FUNCTION_BLOCK "A0301_Spintore_Lat_FB"   // FB59, LAD
TITLE = == GESTIONE DELLA STAZIONE P5 ==
// stored: MemoryReserve 100, SetENOAutomatically false
   VAR_INPUT
      AreaInterface { ExternalAccessible := 'False'; ExternalVisible := 'False'; ExternalWritable := 'False'} : "AreaInterface";
      ZSI { ExternalAccessible := 'False'; ExternalVisible := 'False'; ExternalWritable := 'False'} : "udt_ZoneSafetyInterface";
      DSI { ExternalAccessible := 'False'; ExternalVisible := 'False'; ExternalWritable := 'False'} : "udt_DeviceSafetyInterface";
      DataIn : Struct
         OP_Rest_PB : Bool;
         OP_Work_PB : Bool;
         Orz_1_AnalSens : Int;
         Orz_2_AnalSens : Int;
      END_STRUCT;
      CIn { ExternalAccessible := 'False'; ExternalVisible := 'False'; ExternalWritable := 'False'} : Struct
         Manager_SpinLat_1 : "ValveMachine_Manager";
         Manager_SpinLat_2 : "ValveMachine_Manager";
         Manager_Sollevatori : "ValveMachine_Manager";
         SemiAut_Pb : Bool;
         P4 : Struct
            Fermi : "ValveMachine_COut";
         END_STRUCT;
         P5 : Struct
            SpintoreLong : Struct   // Spintore Longitudinale
               Ax_Sts : Struct
                  PosAttesa_Reached : Bool;
                  PosFineSpinta_Reached : Bool;
               END_STRUCT;
               Spintore : "ValveMachine_COut";
               Ax : "Positioning_EPOS_Machine_COut";
               Vrt : "ValveMachine_COut";
               Orz : "ValveMachine_COut";
            END_STRUCT;
         END_STRUCT;
         Trasporto : "SpeedMachine_COut";
      END_STRUCT;
      Config : Struct
         Vrt_1 : "ValveMachine_Config";
         Orz_1 : "ValveMachine_Config";
         Vrt_2 : "ValveMachine_Config";
         Orz_2 : "ValveMachine_Config";
         Sollevatori : Array[1..7] of "ValveMachine_Config";
         QuotaIngombro_SpinLat2 : Real := 2700.0;
         QuotaIngombro_SpinLat1 { ExternalWritable := 'False'} : Real := 770.0;
         DelayMissingCondition : Time;
      END_STRUCT;
   END_VAR
   VAR_OUTPUT
      MachineInterface : "MachineInterface";
      COut : Struct
         Spin_Lat1 : Struct
            Standstill : Bool;
            Rest_CheckNext : Bool;
            Work_CheckNext : Bool;
            Rest : Bool;
            Work : Bool;
         END_STRUCT;
         Spin_Lat2 : Struct
            Standstill : Bool;
            Rest_CheckNext : Bool;
            Work_CheckNext : Bool;
            Rest : Bool;
            Work : Bool;
         END_STRUCT;
         Vrt_1 : "ValveMachine_COut";
         Orz_1 : "ValveMachine_COut";
         Vrt_2 : "ValveMachine_COut";
         Orz_2 : "ValveMachine_COut";
         Sollevatori : "ValveMachine_COut";
      END_STRUCT;
   END_VAR
   VAR_IN_OUT
      Spin_Lat_1 : Struct
         Par : "Analogic_SensorManagement_Par";
         Data : Struct
            Sens : "Analogic_SensorManagement_Data";
            HMI : "HMI_Preset";
         END_STRUCT;
         Par_Mach : "A0301_Mach_Sens_Par";
      END_STRUCT;
      Spin_Lat_2 : Struct
         Par : "Analogic_SensorManagement_Par";
         Data : Struct
            Sens : "Analogic_SensorManagement_Data";
            HMI : "HMI_Preset";
         END_STRUCT;
         Par_Mach : "A0301_Mach_Sens_Par";
      END_STRUCT;
   END_VAR
   VAR
      Alarm : Struct
         Vrt_1 : "ValveAlr";
         Orz_1 { S7_SetPoint := 'True'} : "ValveAlr";
         Orz_1_AnalSens_Issue : Bool;
         Vrt_2 : "ValveAlr";
         Orz_2 { S7_SetPoint := 'True'} : "ValveAlr";
         Orz_2_AnalSens_Issue : Bool;
         Sollevatori : Array[1..7] of "ValveAlr";
         Finestre : Struct
            SpinLat2_SpinLong_Stop : Bool;   // Allarme Spintore longitudinale a ridosso dello Spintore laterale 2 che non si è abbassato
            SpinLat1_SpinLong_Stop : Bool;   // Allarme Spintore longitudinale a ridosso dello Spintore laterale 1 che non si è abbassato
         END_STRUCT;
      END_STRUCT;
      Warning : Struct
         Vrt_1 : "ValveMachine_Wng";
         Orz_1 { S7_SetPoint := 'True'} : "ValveMachine_Wng";
         Orz_1_AnalSens { ExternalAccessible := 'False'; ExternalVisible := 'False'; ExternalWritable := 'False'} : "Analogic_SensorManagement_Warning";
         Vrt_2 : "ValveMachine_Wng";
         Orz_2 { S7_SetPoint := 'True'} : "ValveMachine_Wng";
         Orz_2_AnalSens { ExternalAccessible := 'False'; ExternalVisible := 'False'; ExternalWritable := 'False'} : "Analogic_SensorManagement_Warning";
         Sollevatori : Array[1..7] of "ValveMachine_Wng";
         Finestre : Struct
            SpinLat2_SpinLong_Stop : Bool;   // Allarme Spintore longitudinale a ridosso dello Spintore laterale 2 che non si è abbassato
            SpinLat1_SpinLong_Stop : Bool;   // Allarme Spintore longitudinale a ridosso dello Spintore laterale 1 che non si è abbassato
         END_STRUCT;
         OP_REST_MissingCnd : Bool;   // Mancanza comando arresto
         OP_WORK_MissingCnd : Bool;   // Mancanza consenso lavoro
      END_STRUCT;
      HMI : Struct
         Selection : Array[1..6] of Bool;   // 0=Disable / 1=Enable Pin
         Sollevatori_Sts { S7_SetPoint := 'True'} : "UDT_HMI-Sts_ValvePosA0301";
         "SpinLat1&2_Sts" { S7_SetPoint := 'True'} : "UDT_HMI-Sts_ValvePosA0301";
         "SpinLat1&2_Vrt_Sts" { S7_SetPoint := 'True'} : "UDT_HMI-Sts_ValvePosA0301";
         "SpinLat1&2_Orz_Sts" { S7_SetPoint := 'True'} : "UDT_HMI-Sts_ValvePosA0301";
         Orz_AnalSens_PB_Preset { ExternalAccessible := 'False'; ExternalVisible := 'False'; ExternalWritable := 'False'} : Bool;   // Pulsante Preset value
         Orz_AnalSens_Preset_Value : LReal;
      END_STRUCT;
      Sts : Struct
         "SpinLat1&2_Alarm" : Bool;
         "SpinLat1&2_Vrt_AlarmPresence" : Bool;
         "SpinLat1&2_Orz_AlarmPresence" : Bool;
         Sollevatori_AlarmPresence : Bool;
         OP_CanMoveFreely : Bool;
         OP_Rest_Cnd : Bool;
         Op_Work_Cnd : Bool;
         Beam : Struct
            H_B : Real;
            Len_Meas : Real;
            P_U_PLen : Real;
            P_L_PLen : Real;
         END_STRUCT;
         "En/Dis_SpinLat_2" : Bool;   // 1=Enable / 0=Disable
      END_STRUCT;
      Ctrl : Struct
         OP_Rest_Man : Bool;
         OP_Work_Man : Bool;
         OP_Rest_Aut : Bool;
         OP_Work_Aut : Bool;
         OP_Rest : Bool;
         OP_Work : Bool;
      END_STRUCT;
      Vrt_1 : "ValveMachine_FB";
      Orz_1 { S7_SetPoint := 'True'} : "ValveMachine_FB";
      Orz_1_AnalSens { S7_SetPoint := 'True'} : "Analogic_SensorManagement";
      Vrt_2 : "ValveMachine_FB";
      Orz_2 { S7_SetPoint := 'True'} : "ValveMachine_FB";
      Orz_2_AnalSens { S7_SetPoint := 'True'} : "Analogic_SensorManagement";
      Sollevatori : Array[1..6] of "ValveMachine_FB";
      AUX : Struct
         OP_Rest_PB : Bool;
         OP_Work_PB : Bool;
      END_STRUCT;
      TON_OP_REST_MissingCnd { S7_SetPoint := 'True'} : TON_TIME;
      TON_OP_WORK_MissingCnd { S7_SetPoint := 'True'} : TON_TIME;
      Finestre : Struct
         Quota_SpinLat2_Rest : Real;   // Quota per comando riposo SpintoreLaterale 2
         Quota_SpinLat1_Rest : Real;   // Quota per comando riposo SpintoreLaterale 1
         RestCnd_Vrt_1 : Bool;   // Spintore longitudinale a ridosso dello Spintore laterale 1 - Comando riposo
         RestCnd_Vrt_2 : Bool;   // Spintore longitudinale a ridosso dello Spintore laterale 2 - Comando riposo
      END_STRUCT;
   END_VAR
   VAR_TEMP
      PE : Struct
         OP_Rest_PB : Bool;
         OP_Work_PB : Bool;
      END_STRUCT;
   END_VAR
   VAR CONSTANT
      Offset_SpinLat2_Rest : Real := 50.0;   // Offset calcolato da quota ingombro Spintore Laterale2 per abbassarlo
      Offset_SpinLat1_Rest : Real := 50.0;   // Offset calcolato da quota ingombro Spintore Laterale1 per abbassarlo
   END_VAR
   VAR_TEMP   // added for the SCL form of the ladder/FBD networks
      _w1 : Bool;
      _w2 : Bool;
      _w3 : Bool;
      _w4 : Bool;
      _w5 : Bool;
      _w6 : Bool;
      _w7 : Bool;
      _w8 : Bool;
   END_VAR
BEGIN

REGION Network 1 (SCL): Reset allarmi
   IF #AreaInterface.RstAlarms THEN
       #Alarm.Orz_1_AnalSens_Issue := FALSE;
       #Alarm.Orz_2_AnalSens_Issue := FALSE;
   END_IF;

   IF #AreaInterface.RstAlarms AND #Vrt_2.COut.Rest AND #Orz_2.COut.Rest THEN
       #Alarm.Finestre.SpinLat2_SpinLong_Stop := 0;
       #Warning.Finestre.SpinLat2_SpinLong_Stop := 0;
   END_IF;

   IF #AreaInterface.RstAlarms AND #Vrt_1.COut.Rest AND #Orz_1.COut.Rest THEN
       #Alarm.Finestre.SpinLat1_SpinLong_Stop := 0;
       #Warning.Finestre.SpinLat1_SpinLong_Stop := 0;
   END_IF;
END_REGION

REGION Network 2: <+>
END_REGION

REGION Network 3: CONTROLLO -
END_REGION

REGION Network 4 (SCL): CONTROLLO - Finestre di ingombro & Controlli di posizione

   // Finestra ingombro SPINTORE LATERALE 2
   #Finestre.Quota_SpinLat2_Rest := #Config.QuotaIngombro_SpinLat2 - #Offset_SpinLat2_Rest;

   // Se ho lo Spintore longitudinale in movimento ed entro dentro la finestra abbasso lo Spintore laterale 2 prima di arrivarci addosso
   // //
   IF #Sts.Beam.Len_Meas <= 2700.0 THEN
       #Sts."En/Dis_SpinLat_2" := FALSE;

   ELSE
       #Sts."En/Dis_SpinLat_2" := TRUE;
       #Warning.Finestre.SpinLat2_SpinLong_Stop := FALSE;
   END_IF;

   //Se arrivo in quota ingombro spintore lat. 2 mando a riposo attivando il cmd finestra
   IF  #Finestre.Quota_SpinLat2_Rest <= #CIn.P5.SpintoreLong.Ax.ActualPosition THEN
       #Finestre.RestCnd_Vrt_2 := TRUE;
   ELSE
       #Finestre.RestCnd_Vrt_2 := FALSE;
   END_IF;

   // Se supero la quota di riposo Spintore Laterale 2 e non sono ancora a riposo con Spintore Laterale attivo warning
   IF #Finestre.Quota_SpinLat2_Rest < #CIn.P5.SpintoreLong.Ax.ActualPosition AND NOT #Vrt_2.COut.Rest THEN
       #Warning.Finestre.SpinLat2_SpinLong_Stop := TRUE;
   END_IF;

   //Se vado a riposo con spin. lat 2 resetto warning 
   IF (#Vrt_2.COut.Rest AND #Orz_2.COut.Rest) THEN
       #Warning.Finestre.SpinLat2_SpinLong_Stop := FALSE;
   END_IF;

   // Finestra ingombro SPINTORE LATERALE 1
   #Finestre.Quota_SpinLat1_Rest := #Config.QuotaIngombro_SpinLat1 - #Offset_SpinLat1_Rest;

   // Se ho lo Spintore longitudinale in movimento ed entro dentro la finestra abbasso lo Spintore laterale 1 prima di arrivarci addosso

   //Se arrivo in quota ingombro spintore lat. 1 mando a riposo attivando il cmd finestra 
   IF #Finestre.Quota_SpinLat1_Rest <= #CIn.P5.SpintoreLong.Ax.ActualPosition  THEN
       #Finestre.RestCnd_Vrt_1 := TRUE;
   ELSE
       #Finestre.RestCnd_Vrt_1 := FALSE;
   END_IF;

   // Se supero la quota di riposo Spintore Laterale 1 e non sono ancora a riposo con Spintore Laterale attivo warning
   IF #Finestre.Quota_SpinLat1_Rest < #CIn.P5.SpintoreLong.Ax.ActualPosition AND NOT #Vrt_1.COut.Rest THEN
       #Warning.Finestre.SpinLat1_SpinLong_Stop := TRUE;
   END_IF;

   //Se vado a riposo con spin. lat 2 resetto warning 
   IF (#Vrt_1.COut.Rest AND #Orz_1.COut.Rest) THEN
       #Warning.Finestre.SpinLat2_SpinLong_Stop := FALSE;

   END_IF;
END_REGION

REGION Network 5: <+>
END_REGION

REGION Network 6: Operazione può muoversi liberamente perchè non sposta nessun BEAM
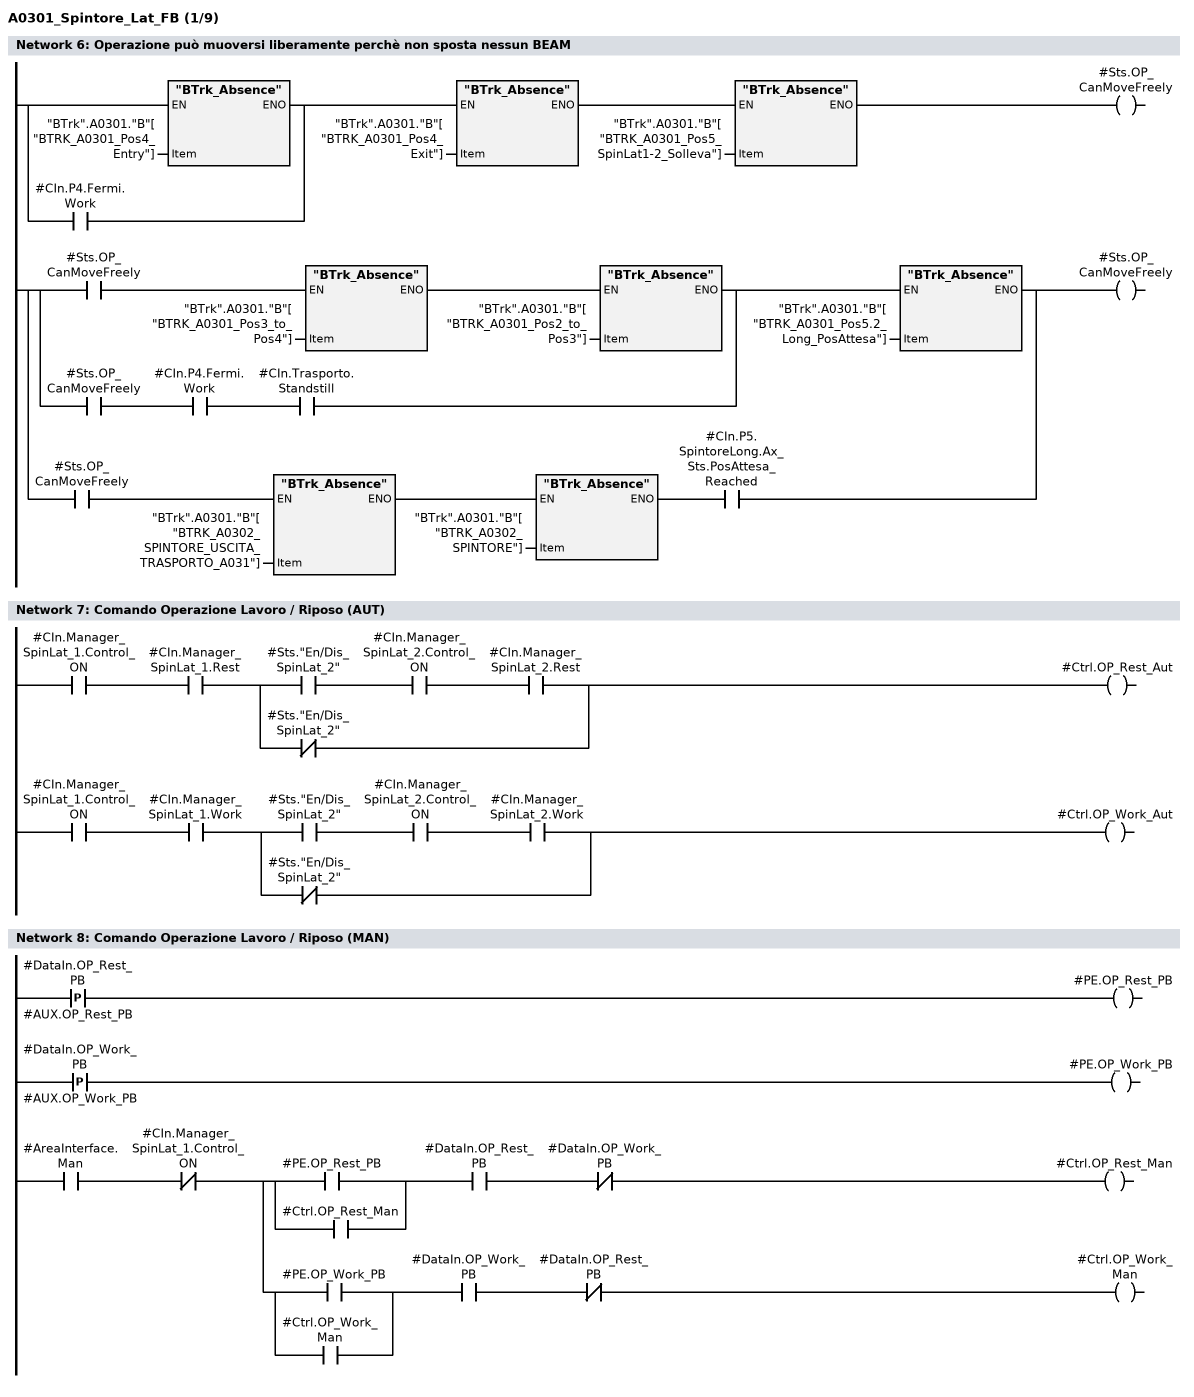
   RUNG wire#powerrail
      "BTrk_Absence"(Item := "BTrk".A0301."B"["BTRK_A0301_Pos4_Entry"])
      wire#w1
      "BTrk_Absence"(Item := "BTrk".A0301."B"["BTRK_A0301_Pos4_Exit"])
      "BTrk_Absence"(Item := "BTrk".A0301."B"["BTRK_A0301_Pos5_SpinLat1-2_Solleva"])
      Coil( #Sts.OP_CanMoveFreely )
   END_RUNG
   RUNG wire#powerrail
      Contact( #CIn.P4.Fermi.Work )
   END_RUNG wire#w1
   RUNG wire#powerrail
      Contact( #Sts.OP_CanMoveFreely )
      "BTrk_Absence"(Item := "BTrk".A0301."B"["BTRK_A0301_Pos3_to_Pos4"])
      "BTrk_Absence"(Item := "BTrk".A0301."B"["BTRK_A0301_Pos2_to_Pos3"])
      wire#w2
      "BTrk_Absence"(Item := "BTrk".A0301."B"["BTRK_A0301_Pos5.2_Long_PosAttesa"])
      wire#w3
      Coil( #Sts.OP_CanMoveFreely )
   END_RUNG
   RUNG wire#powerrail
      Contact( #Sts.OP_CanMoveFreely )
      Contact( #CIn.P4.Fermi.Work )
      Contact( #CIn.Trasporto.Standstill )
   END_RUNG wire#w2
   RUNG wire#powerrail
      Contact( #Sts.OP_CanMoveFreely )
      "BTrk_Absence"(Item := "BTrk".A0301."B"["BTRK_A0302_SPINTORE_USCITA_TRASPORTO_A031"])
      "BTrk_Absence"(Item := "BTrk".A0301."B"["BTRK_A0302_SPINTORE"])
      Contact( #CIn.P5.SpintoreLong.Ax_Sts.PosAttesa_Reached )
   END_RUNG wire#w3
   // the same network as SCL:
   "BTrk_Absence"(Item := "BTrk".A0301."B"["BTRK_A0301_Pos4_Entry"], ENO => #_w1);
   "BTrk_Absence"(EN := #_w1 OR #CIn.P4.Fermi.Work,
                  Item := "BTrk".A0301."B"["BTRK_A0301_Pos4_Exit"],
                  ENO => #_w2);
   "BTrk_Absence"(EN := #_w2, Item := "BTrk".A0301."B"["BTRK_A0301_Pos5_SpinLat1-2_Solleva"], ENO => #_w3);
   #Sts.OP_CanMoveFreely := #_w3;
   "BTrk_Absence"(EN := #Sts.OP_CanMoveFreely, Item := "BTrk".A0301."B"["BTRK_A0301_Pos3_to_Pos4"], ENO => #_w4);
   "BTrk_Absence"(EN := #_w4, Item := "BTrk".A0301."B"["BTRK_A0301_Pos2_to_Pos3"], ENO => #_w5);
   "BTrk_Absence"(EN := #_w5 OR (#Sts.OP_CanMoveFreely AND #CIn.P4.Fermi.Work AND #CIn.Trasporto.Standstill),
                  Item := "BTrk".A0301."B"["BTRK_A0301_Pos5.2_Long_PosAttesa"],
                  ENO => #_w6);
   "BTrk_Absence"(EN := #Sts.OP_CanMoveFreely,
                  Item := "BTrk".A0301."B"["BTRK_A0302_SPINTORE_USCITA_TRASPORTO_A031"],
                  ENO => #_w7);
   "BTrk_Absence"(EN := #_w7, Item := "BTrk".A0301."B"["BTRK_A0302_SPINTORE"], ENO => #_w8);
   #Sts.OP_CanMoveFreely := #_w6 OR (#_w8 AND #CIn.P5.SpintoreLong.Ax_Sts.PosAttesa_Reached);
END_REGION

REGION Network 7: Comando Operazione Lavoro / Riposo (AUT)
   RUNG wire#powerrail
      Contact( #CIn.Manager_SpinLat_1.Control_ON )
      Contact( #CIn.Manager_SpinLat_1.Rest )
      wire#w1
      Contact( #Sts."En/Dis_SpinLat_2" )
      Contact( #CIn.Manager_SpinLat_2.Control_ON )
      Contact( #CIn.Manager_SpinLat_2.Rest )
      wire#w2
      Coil( #Ctrl.OP_Rest_Aut )
   END_RUNG
   RUNG wire#w1
      I_Contact( #Sts."En/Dis_SpinLat_2" )
   END_RUNG wire#w2
   RUNG wire#powerrail
      Contact( #CIn.Manager_SpinLat_1.Control_ON )
      Contact( #CIn.Manager_SpinLat_1.Work )
      wire#w3
      Contact( #Sts."En/Dis_SpinLat_2" )
      Contact( #CIn.Manager_SpinLat_2.Control_ON )
      Contact( #CIn.Manager_SpinLat_2.Work )
      wire#w4
      Coil( #Ctrl.OP_Work_Aut )
   END_RUNG
   RUNG wire#w3
      I_Contact( #Sts."En/Dis_SpinLat_2" )
   END_RUNG wire#w4
   // the same network as SCL:
   #Ctrl.OP_Rest_Aut := #CIn.Manager_SpinLat_1.Control_ON AND #CIn.Manager_SpinLat_1.Rest AND ((#Sts."En/Dis_SpinLat_2" AND #CIn.Manager_SpinLat_2.Control_ON AND #CIn.Manager_SpinLat_2.Rest) OR NOT #Sts."En/Dis_SpinLat_2");
   #Ctrl.OP_Work_Aut := #CIn.Manager_SpinLat_1.Control_ON AND #CIn.Manager_SpinLat_1.Work AND ((#Sts."En/Dis_SpinLat_2" AND #CIn.Manager_SpinLat_2.Control_ON AND #CIn.Manager_SpinLat_2.Work) OR NOT #Sts."En/Dis_SpinLat_2");
END_REGION

REGION Network 8: Comando Operazione Lavoro / Riposo (MAN)
   RUNG wire#powerrail
      P_Contact(operand := #DataIn.OP_Rest_PB, bit := #AUX.OP_Rest_PB)
      Coil( #PE.OP_Rest_PB )
   END_RUNG
   RUNG wire#powerrail
      P_Contact(operand := #DataIn.OP_Work_PB, bit := #AUX.OP_Work_PB)
      Coil( #PE.OP_Work_PB )
   END_RUNG
   RUNG wire#powerrail
      Contact( #AreaInterface.Man )
      I_Contact( #CIn.Manager_SpinLat_1.Control_ON )
      wire#w1
      Contact( #PE.OP_Rest_PB )
      wire#w2
      Contact( #DataIn.OP_Rest_PB )
      I_Contact( #DataIn.OP_Work_PB )
      Coil( #Ctrl.OP_Rest_Man )
   END_RUNG
   RUNG wire#w1
      Contact( #Ctrl.OP_Rest_Man )
   END_RUNG wire#w2
   RUNG wire#w1
      Contact( #PE.OP_Work_PB )
      wire#w3
      Contact( #DataIn.OP_Work_PB )
      I_Contact( #DataIn.OP_Rest_PB )
      Coil( #Ctrl.OP_Work_Man )
   END_RUNG
   RUNG wire#w1
      Contact( #Ctrl.OP_Work_Man )
   END_RUNG wire#w3
   // the same network as SCL:
   #_w1 := #DataIn.OP_Rest_PB AND NOT #AUX.OP_Rest_PB;   // rising edge of #DataIn.OP_Rest_PB
   #AUX.OP_Rest_PB := #DataIn.OP_Rest_PB;
   #PE.OP_Rest_PB := #_w1;
   #_w2 := #DataIn.OP_Work_PB AND NOT #AUX.OP_Work_PB;   // rising edge of #DataIn.OP_Work_PB
   #AUX.OP_Work_PB := #DataIn.OP_Work_PB;
   #PE.OP_Work_PB := #_w2;
   #_w3 := #AreaInterface.Man AND NOT #CIn.Manager_SpinLat_1.Control_ON;
   #Ctrl.OP_Rest_Man := #_w3 AND (#PE.OP_Rest_PB OR #Ctrl.OP_Rest_Man) AND #DataIn.OP_Rest_PB AND NOT #DataIn.OP_Work_PB;
   #Ctrl.OP_Work_Man := #_w3 AND (#PE.OP_Work_PB OR #Ctrl.OP_Work_Man) AND #DataIn.OP_Work_PB AND NOT #DataIn.OP_Rest_PB;
END_REGION

REGION Network 9: Cumulativo Operazione Lavoro / Riposo (ALL)
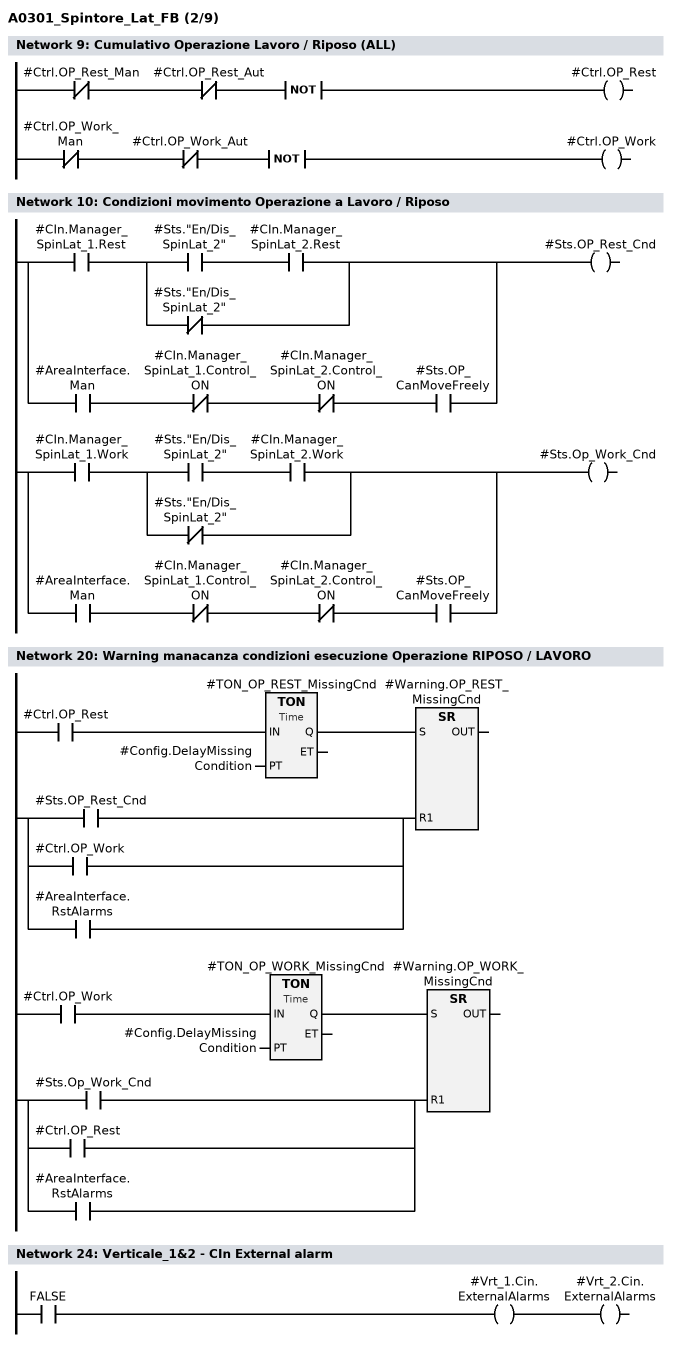
   RUNG wire#powerrail
      I_Contact( #Ctrl.OP_Rest_Man )
      I_Contact( #Ctrl.OP_Rest_Aut )
      Not()
      Coil( #Ctrl.OP_Rest )
   END_RUNG
   RUNG wire#powerrail
      I_Contact( #Ctrl.OP_Work_Man )
      I_Contact( #Ctrl.OP_Work_Aut )
      Not()
      Coil( #Ctrl.OP_Work )
   END_RUNG
   // the same network as SCL:
   #Ctrl.OP_Rest := NOT (NOT #Ctrl.OP_Rest_Man AND NOT #Ctrl.OP_Rest_Aut);
   #Ctrl.OP_Work := NOT (NOT #Ctrl.OP_Work_Man AND NOT #Ctrl.OP_Work_Aut);
END_REGION

REGION Network 10: Condizioni movimento Operazione a Lavoro / Riposo
   RUNG wire#powerrail
      Contact( #CIn.Manager_SpinLat_1.Rest )
      wire#w1
      Contact( #Sts."En/Dis_SpinLat_2" )
      Contact( #CIn.Manager_SpinLat_2.Rest )
      wire#w2
      Coil( #Sts.OP_Rest_Cnd )
   END_RUNG
   RUNG wire#w1
      I_Contact( #Sts."En/Dis_SpinLat_2" )
   END_RUNG wire#w2
   RUNG wire#powerrail
      Contact( #AreaInterface.Man )
      I_Contact( #CIn.Manager_SpinLat_1.Control_ON )
      I_Contact( #CIn.Manager_SpinLat_2.Control_ON )
      Contact( #Sts.OP_CanMoveFreely )
   END_RUNG wire#w2
   RUNG wire#powerrail
      Contact( #CIn.Manager_SpinLat_1.Work )
      wire#w3
      Contact( #Sts."En/Dis_SpinLat_2" )
      Contact( #CIn.Manager_SpinLat_2.Work )
      wire#w4
      Coil( #Sts.Op_Work_Cnd )
   END_RUNG
   RUNG wire#w3
      I_Contact( #Sts."En/Dis_SpinLat_2" )
   END_RUNG wire#w4
   RUNG wire#powerrail
      Contact( #AreaInterface.Man )
      I_Contact( #CIn.Manager_SpinLat_1.Control_ON )
      I_Contact( #CIn.Manager_SpinLat_2.Control_ON )
      Contact( #Sts.OP_CanMoveFreely )
   END_RUNG wire#w4
   // the same network as SCL:
   #Sts.OP_Rest_Cnd := (#CIn.Manager_SpinLat_1.Rest AND ((#Sts."En/Dis_SpinLat_2" AND #CIn.Manager_SpinLat_2.Rest) OR NOT #Sts."En/Dis_SpinLat_2")) OR (#AreaInterface.Man AND NOT #CIn.Manager_SpinLat_1.Control_ON AND NOT #CIn.Manager_SpinLat_2.Control_ON AND #Sts.OP_CanMoveFreely);
   #Sts.Op_Work_Cnd := (#CIn.Manager_SpinLat_1.Work AND ((#Sts."En/Dis_SpinLat_2" AND #CIn.Manager_SpinLat_2.Work) OR NOT #Sts."En/Dis_SpinLat_2")) OR (#AreaInterface.Man AND NOT #CIn.Manager_SpinLat_1.Control_ON AND NOT #CIn.Manager_SpinLat_2.Control_ON AND #Sts.OP_CanMoveFreely);
END_REGION

REGION Network 11: <+>
END_REGION

REGION Network 12 (SCL): Verticale + Orizzontale 1 - Cin Manager (Esecuzione sequenza comandi)
   #Vrt_1.Cin.Manager.Control_ON := #Orz_1.Cin.Manager.Control_ON := #CIn.Manager_SpinLat_1.Control_ON;

   #Vrt_1.Cin.Manager.Rest := FALSE;
   #Vrt_1.Cin.Manager.Work := FALSE;
   #Orz_1.Cin.Manager.Rest := FALSE;
   #Orz_1.Cin.Manager.Work := FALSE;


       IF (#Ctrl.OP_Rest AND #Sts.OP_Rest_Cnd) OR #Finestre.RestCnd_Vrt_1 THEN

           #Orz_1.Cin.Manager.Rest := #Vrt_1.Cin.Manager.Rest := TRUE;

       ELSIF (#Ctrl.OP_Work AND #Sts.Op_Work_Cnd) AND NOT #Finestre.RestCnd_Vrt_1 THEN

           #Orz_1.Cin.Manager.Work := #Vrt_1.Cin.Manager.Work := TRUE;

       END_IF;
END_REGION

REGION Network 13 (SCL): Verticale + Orizzontale1 - CIn Abilitazioni Stop Manager
   #Vrt_1.Cin.Manager.EnableStopDoorOpeningReq := #Orz_1.Cin.Manager.EnableStopDoorOpeningReq := #CIn.Manager_SpinLat_1.EnableStopDoorOpeningReq;

   #Vrt_1.Cin.Manager.EnableStopInPhase := #Orz_1.Cin.Manager.EnableStopInPhase := #CIn.Manager_SpinLat_1.EnableStopInPhase;

   #Vrt_1.Cin.Manager.EnableStopProgrammed := #Orz_1.Cin.Manager.EnableStopProgrammed := #CIn.Manager_SpinLat_1.EnableStopProgrammed;
END_REGION

REGION Network 14 (SCL): Verticale + Orizzontale 2 - Cin Manager (Esecuzione sequenza comandi)
   // Controllo della misura in lunghezza del Beam per sapere se abilitare il secondo spintore
   //
   #Vrt_2.Cin.Manager.Control_ON := #Orz_2.Cin.Manager.Control_ON := #CIn.Manager_SpinLat_2.Control_ON;
   //
   #Vrt_2.Cin.Manager.Rest := FALSE;
   #Vrt_2.Cin.Manager.Work := FALSE;
   #Orz_2.Cin.Manager.Rest := FALSE;
   #Orz_2.Cin.Manager.Work := FALSE;



   IF (#Ctrl.OP_Rest AND #Sts.OP_Rest_Cnd )OR #Finestre.RestCnd_Vrt_2 OR #Warning.Finestre.SpinLat2_SpinLong_Stop THEN

           #Orz_2.Cin.Manager.Rest := #Vrt_2.Cin.Manager.Rest := TRUE;

       ELSIF (#Ctrl.OP_Work AND #Sts.Op_Work_Cnd) AND #Sts."En/Dis_SpinLat_2" AND NOT #Finestre.RestCnd_Vrt_2  THEN

           #Orz_2.Cin.Manager.Work := #Vrt_2.Cin.Manager.Work := TRUE;

       END_IF;
END_REGION

REGION Network 15 (SCL): Verticale + Orizzontale 2 - CIn Abilitazioni Stop Manager
   #Vrt_2.Cin.Manager.EnableStopDoorOpeningReq := #Orz_2.Cin.Manager.EnableStopDoorOpeningReq := #CIn.Manager_SpinLat_2.EnableStopDoorOpeningReq;

   #Vrt_2.Cin.Manager.EnableStopInPhase := #Orz_2.Cin.Manager.EnableStopInPhase := #CIn.Manager_SpinLat_2.EnableStopInPhase;

   #Vrt_2.Cin.Manager.EnableStopProgrammed := #Orz_2.Cin.Manager.EnableStopProgrammed := #CIn.Manager_SpinLat_2.EnableStopProgrammed;
END_REGION

REGION Network 16: <+>
END_REGION

REGION Network 17 (SCL): S[1...7] Sollevatori - Cin Manager Comando arresto / lavoro
   //
   #Sollevatori[1].Cin.Manager.Rest := FALSE;
   #Sollevatori[2].Cin.Manager.Rest := FALSE;
   #Sollevatori[3].Cin.Manager.Rest := FALSE;
   #Sollevatori[4].Cin.Manager.Rest := FALSE;
   #Sollevatori[5].Cin.Manager.Rest := FALSE;
   #Sollevatori[6].Cin.Manager.Rest := FALSE;
   //************************************
   #Sollevatori[1].Cin.Manager.Work := FALSE;
   #Sollevatori[2].Cin.Manager.Work := FALSE;
   #Sollevatori[3].Cin.Manager.Work := FALSE;
   #Sollevatori[4].Cin.Manager.Work := FALSE;
   #Sollevatori[5].Cin.Manager.Work := FALSE;
   #Sollevatori[6].Cin.Manager.Work := FALSE;
   //
   // CIn Manager  Control ON se ho un richiesta di comando attiva
   IF #AreaInterface.Aut OR #CIn.SemiAut_Pb THEN
       #Sollevatori[1].Cin.Manager.Control_ON := TRUE;
       #Sollevatori[2].Cin.Manager.Control_ON := TRUE;
       #Sollevatori[3].Cin.Manager.Control_ON := TRUE;
       #Sollevatori[4].Cin.Manager.Control_ON := TRUE;
       #Sollevatori[5].Cin.Manager.Control_ON := TRUE;
       #Sollevatori[6].Cin.Manager.Control_ON := TRUE;
   ELSE
       #Sollevatori[1].Cin.Manager.Control_ON := FALSE;
       #Sollevatori[2].Cin.Manager.Control_ON := FALSE;
       #Sollevatori[3].Cin.Manager.Control_ON := FALSE;
       #Sollevatori[4].Cin.Manager.Control_ON := FALSE;
       #Sollevatori[5].Cin.Manager.Control_ON := FALSE;
       #Sollevatori[6].Cin.Manager.Control_ON := FALSE;
   END_IF;

   // CIn Manager Rest se ho un richiesta di comando arresto attiva
   IF #CIn.Manager_Sollevatori.Rest THEN

       #Sollevatori[1].Cin.Manager.Rest := TRUE;
       #Sollevatori[2].Cin.Manager.Rest := TRUE;
       #Sollevatori[3].Cin.Manager.Rest := TRUE;
       #Sollevatori[4].Cin.Manager.Rest := TRUE;
       #Sollevatori[5].Cin.Manager.Rest := TRUE;
       #Sollevatori[6].Cin.Manager.Rest := TRUE;

       // CIn Manager Work se ho un richiesta di comando lavoro attiva   
       ELSIF #CIn.Manager_Sollevatori.Work THEN

       #Sollevatori[1].Cin.Manager.Work := TRUE;
       #Sollevatori[2].Cin.Manager.Work := TRUE;
       #Sollevatori[3].Cin.Manager.Work := TRUE;
       #Sollevatori[4].Cin.Manager.Work := TRUE;
       #Sollevatori[5].Cin.Manager.Work := TRUE;
       #Sollevatori[6].Cin.Manager.Work := TRUE;

   END_IF;
END_REGION

REGION Network 18 (SCL): S[1...7] Sollevatori - CIn Abilitazioni Stop Manager
   //
   // CIn Manager Stop per richiesta apertura safety
   IF #CIn.Manager_SpinLat_1.EnableStopDoorOpeningReq THEN
       #Sollevatori[1].Cin.Manager.EnableStopDoorOpeningReq := TRUE;
       #Sollevatori[2].Cin.Manager.EnableStopDoorOpeningReq := TRUE;
       #Sollevatori[3].Cin.Manager.EnableStopDoorOpeningReq := TRUE;
       #Sollevatori[4].Cin.Manager.EnableStopDoorOpeningReq := TRUE;
       #Sollevatori[5].Cin.Manager.EnableStopDoorOpeningReq := TRUE;
       #Sollevatori[6].Cin.Manager.EnableStopDoorOpeningReq := TRUE;

   ELSE
       #Sollevatori[1].Cin.Manager.EnableStopDoorOpeningReq := FALSE;
       #Sollevatori[2].Cin.Manager.EnableStopDoorOpeningReq := FALSE;
       #Sollevatori[3].Cin.Manager.EnableStopDoorOpeningReq := FALSE;
       #Sollevatori[4].Cin.Manager.EnableStopDoorOpeningReq := FALSE;
       #Sollevatori[5].Cin.Manager.EnableStopDoorOpeningReq := FALSE;
       #Sollevatori[6].Cin.Manager.EnableStopDoorOpeningReq := FALSE;

   END_IF;
   // CIn Manager Stop in fase delle macchine precedenti
   IF #CIn.Manager_SpinLat_1.EnableStopInPhase THEN
       #Sollevatori[1].Cin.Manager.EnableStopInPhase := TRUE;
       #Sollevatori[2].Cin.Manager.EnableStopInPhase := TRUE;
       #Sollevatori[3].Cin.Manager.EnableStopInPhase := TRUE;
       #Sollevatori[4].Cin.Manager.EnableStopInPhase := TRUE;
       #Sollevatori[5].Cin.Manager.EnableStopInPhase := TRUE;
       #Sollevatori[6].Cin.Manager.EnableStopInPhase := TRUE;

   ELSE
       #Sollevatori[1].Cin.Manager.EnableStopInPhase := FALSE;
       #Sollevatori[2].Cin.Manager.EnableStopInPhase := FALSE;
       #Sollevatori[3].Cin.Manager.EnableStopInPhase := FALSE;
       #Sollevatori[4].Cin.Manager.EnableStopInPhase := FALSE;
       #Sollevatori[5].Cin.Manager.EnableStopInPhase := FALSE;
       #Sollevatori[6].Cin.Manager.EnableStopInPhase := FALSE;

   END_IF;

   // CIn Manager Stop programmato configurabile a piacere
   IF #CIn.Manager_SpinLat_1.EnableStopProgrammed THEN
       #Sollevatori[1].Cin.Manager.EnableStopProgrammed := TRUE;
       #Sollevatori[2].Cin.Manager.EnableStopProgrammed := TRUE;
       #Sollevatori[3].Cin.Manager.EnableStopProgrammed := TRUE;
       #Sollevatori[4].Cin.Manager.EnableStopProgrammed := TRUE;
       #Sollevatori[5].Cin.Manager.EnableStopProgrammed := TRUE;
       #Sollevatori[6].Cin.Manager.EnableStopProgrammed := TRUE;

   ELSE
       #Sollevatori[1].Cin.Manager.EnableStopProgrammed := FALSE;
       #Sollevatori[2].Cin.Manager.EnableStopProgrammed := FALSE;
       #Sollevatori[3].Cin.Manager.EnableStopProgrammed := FALSE;
       #Sollevatori[4].Cin.Manager.EnableStopProgrammed := FALSE;
       #Sollevatori[5].Cin.Manager.EnableStopProgrammed := FALSE;
       #Sollevatori[6].Cin.Manager.EnableStopProgrammed := FALSE;

   END_IF;
END_REGION

REGION Network 19: <+>
END_REGION

REGION Network 20: Warning manacanza condizioni esecuzione Operazione RIPOSO / LAVORO
   RUNG wire#powerrail
      Contact( #Ctrl.OP_Rest )
      { S7_Templates := "time_type := Time" } #TON_OP_REST_MissingCnd.TON(pt := #Config.DelayMissingCondition, et =>)
      S_SR(operand := #Warning.OP_REST_MissingCnd, r1 := wire#w1)
   END_RUNG
   RUNG wire#powerrail
      Contact( #Sts.OP_Rest_Cnd )
   END_RUNG wire#w1
   RUNG wire#powerrail
      Contact( #Ctrl.OP_Work )
   END_RUNG wire#w1
   RUNG wire#powerrail
      Contact( #AreaInterface.RstAlarms )
   END_RUNG wire#w1
   RUNG wire#powerrail
      Contact( #Ctrl.OP_Work )
      { S7_Templates := "time_type := Time" } #TON_OP_WORK_MissingCnd.TON(pt := #Config.DelayMissingCondition, et =>)
      S_SR(operand := #Warning.OP_WORK_MissingCnd, r1 := wire#w2)
   END_RUNG
   RUNG wire#powerrail
      Contact( #Sts.Op_Work_Cnd )
   END_RUNG wire#w2
   RUNG wire#powerrail
      Contact( #Ctrl.OP_Rest )
   END_RUNG wire#w2
   RUNG wire#powerrail
      Contact( #AreaInterface.RstAlarms )
   END_RUNG wire#w2
   // the same network as SCL:
   #TON_OP_REST_MissingCnd(IN := #Ctrl.OP_Rest, PT := #Config.DelayMissingCondition);   // TON
   IF #TON_OP_REST_MissingCnd.Q THEN
       #Warning.OP_REST_MissingCnd := TRUE;   // SR flip-flop
   END_IF;
   IF #Sts.OP_Rest_Cnd OR #Ctrl.OP_Work OR #AreaInterface.RstAlarms THEN
       #Warning.OP_REST_MissingCnd := FALSE;
   END_IF;
   #TON_OP_WORK_MissingCnd(IN := #Ctrl.OP_Work, PT := #Config.DelayMissingCondition);   // TON
   IF #TON_OP_WORK_MissingCnd.Q THEN
       #Warning.OP_WORK_MissingCnd := TRUE;   // SR flip-flop
   END_IF;
   IF #Sts.Op_Work_Cnd OR #Ctrl.OP_Rest OR #AreaInterface.RstAlarms THEN
       #Warning.OP_WORK_MissingCnd := FALSE;
   END_IF;
END_REGION

REGION Network 21: <+>
END_REGION

REGION Network 22: << GESTIONE VERTICALE >>
END_REGION

REGION Network 23 (SCL): Verticale1&2 - Data In
   // DataIn Scritti sulla CALL dell'FB
END_REGION

REGION Network 24: Verticale_1&2 - CIn External alarm
   RUNG wire#powerrail
      Contact( FALSE )
      Coil( #Vrt_1.Cin.ExternalAlarms )
      Coil( #Vrt_2.Cin.ExternalAlarms )
   END_RUNG
   // the same network as SCL:
   #Vrt_1.Cin.ExternalAlarms := FALSE;
   #Vrt_2.Cin.ExternalAlarms := FALSE;
END_REGION

REGION Network 25: Verticale_1 - Cin Ext Enable
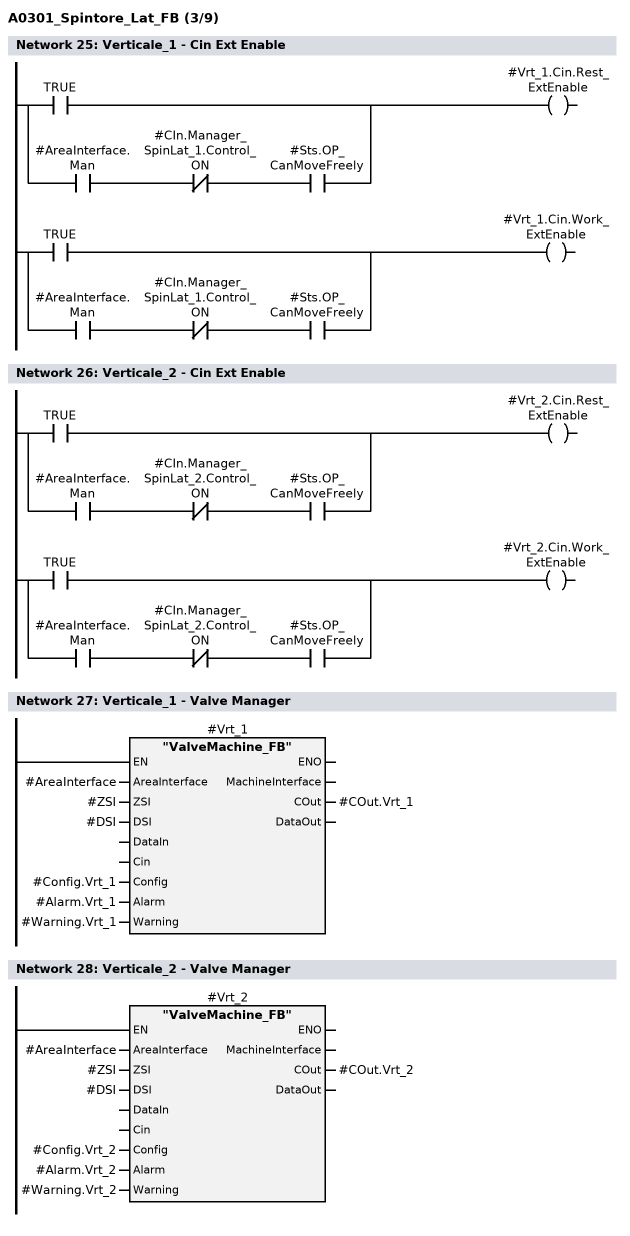
   RUNG wire#powerrail
      Contact( TRUE )
      wire#w1
      Coil( #Vrt_1.Cin.Rest_ExtEnable )
   END_RUNG
   RUNG wire#powerrail
      Contact( #AreaInterface.Man )
      I_Contact( #CIn.Manager_SpinLat_1.Control_ON )
      Contact( #Sts.OP_CanMoveFreely )
   END_RUNG wire#w1
   RUNG wire#powerrail
      Contact( TRUE )
      wire#w2
      Coil( #Vrt_1.Cin.Work_ExtEnable )
   END_RUNG
   RUNG wire#powerrail
      Contact( #AreaInterface.Man )
      I_Contact( #CIn.Manager_SpinLat_1.Control_ON )
      Contact( #Sts.OP_CanMoveFreely )
   END_RUNG wire#w2
   // the same network as SCL:
   #Vrt_1.Cin.Rest_ExtEnable := TRUE OR (#AreaInterface.Man AND NOT #CIn.Manager_SpinLat_1.Control_ON AND #Sts.OP_CanMoveFreely);
   #Vrt_1.Cin.Work_ExtEnable := TRUE OR (#AreaInterface.Man AND NOT #CIn.Manager_SpinLat_1.Control_ON AND #Sts.OP_CanMoveFreely);
END_REGION

REGION Network 26: Verticale_2 - Cin Ext Enable
   RUNG wire#powerrail
      Contact( TRUE )
      wire#w1
      Coil( #Vrt_2.Cin.Rest_ExtEnable )
   END_RUNG
   RUNG wire#powerrail
      Contact( #AreaInterface.Man )
      I_Contact( #CIn.Manager_SpinLat_2.Control_ON )
      Contact( #Sts.OP_CanMoveFreely )
   END_RUNG wire#w1
   RUNG wire#powerrail
      Contact( TRUE )
      wire#w2
      Coil( #Vrt_2.Cin.Work_ExtEnable )
   END_RUNG
   RUNG wire#powerrail
      Contact( #AreaInterface.Man )
      I_Contact( #CIn.Manager_SpinLat_2.Control_ON )
      Contact( #Sts.OP_CanMoveFreely )
   END_RUNG wire#w2
   // the same network as SCL:
   #Vrt_2.Cin.Rest_ExtEnable := TRUE OR (#AreaInterface.Man AND NOT #CIn.Manager_SpinLat_2.Control_ON AND #Sts.OP_CanMoveFreely);
   #Vrt_2.Cin.Work_ExtEnable := TRUE OR (#AreaInterface.Man AND NOT #CIn.Manager_SpinLat_2.Control_ON AND #Sts.OP_CanMoveFreely);
END_REGION

REGION Network 27: Verticale_1 - Valve Manager
   RUNG wire#powerrail
      #Vrt_1(AreaInterface := #AreaInterface, ZSI := #ZSI, DSI := #DSI, DataIn :=, Cin :=, Config := #Config.Vrt_1, Alarm := #Alarm.Vrt_1, Warning := #Warning.Vrt_1, MachineInterface =>, COut => #COut.Vrt_1, DataOut =>)
   END_RUNG
   // the same network as SCL:
   #Vrt_1(AreaInterface := #AreaInterface,   // "ValveMachine_FB"
          ZSI := #ZSI,
          DSI := #DSI,
          Config := #Config.Vrt_1,
          Alarm := #Alarm.Vrt_1,
          Warning := #Warning.Vrt_1,
          COut => #COut.Vrt_1);
END_REGION

REGION Network 28: Verticale_2 - Valve Manager
   RUNG wire#powerrail
      #Vrt_2(AreaInterface := #AreaInterface, ZSI := #ZSI, DSI := #DSI, DataIn :=, Cin :=, Config := #Config.Vrt_2, Alarm := #Alarm.Vrt_2, Warning := #Warning.Vrt_2, MachineInterface =>, COut => #COut.Vrt_2, DataOut =>)
   END_RUNG
   // the same network as SCL:
   #Vrt_2(AreaInterface := #AreaInterface,   // "ValveMachine_FB"
          ZSI := #ZSI,
          DSI := #DSI,
          Config := #Config.Vrt_2,
          Alarm := #Alarm.Vrt_2,
          Warning := #Warning.Vrt_2,
          COut => #COut.Vrt_2);
END_REGION

REGION Network 29: << GESTIONE ORIZZONTALE >>
END_REGION

REGION Network 30: <+>
END_REGION

REGION Network 31: << GESTIONE SPINTORE ORIZZ_1&2 - ANALOGIC SENSOR >>
END_REGION

REGION Network 33: Orizzontale_1 -Scalatura sensore
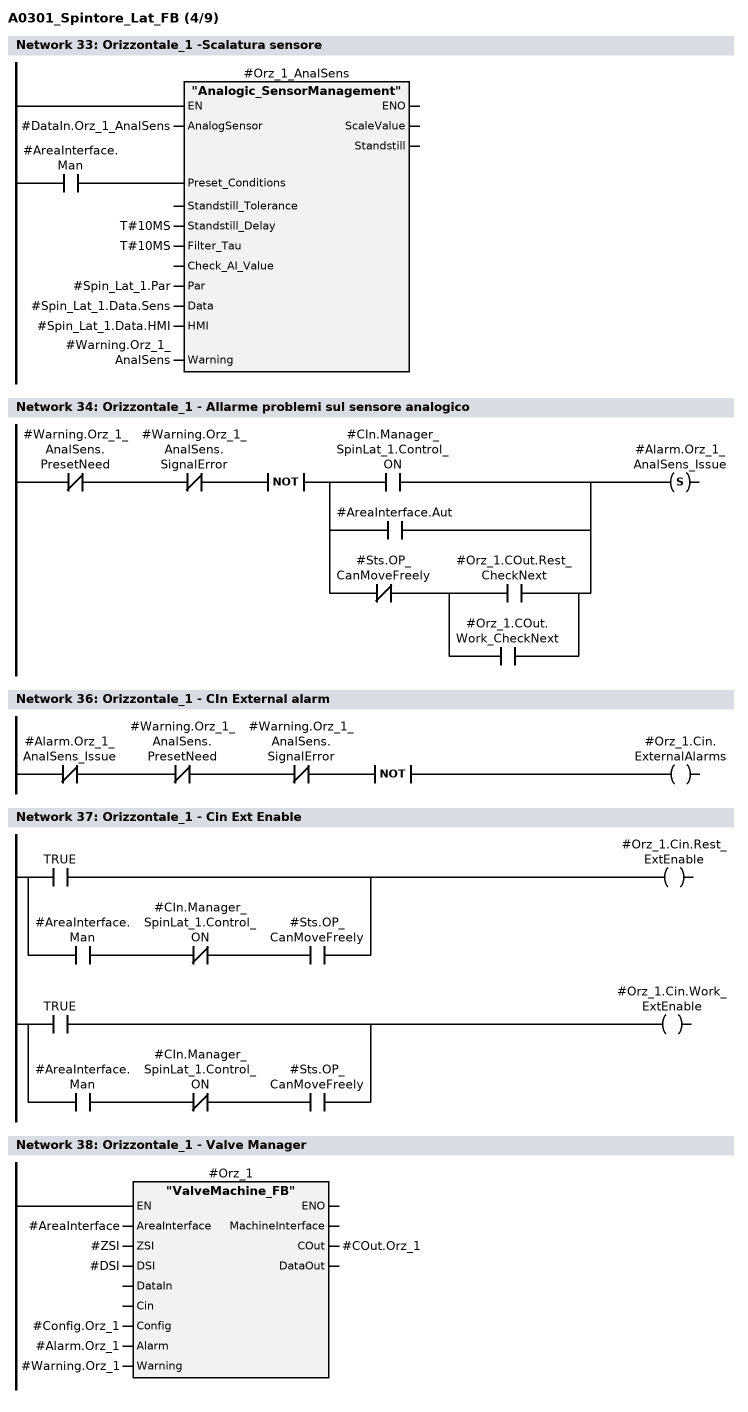
   RUNG wire#powerrail
      #Orz_1_AnalSens(Preset_Conditions := wire#w1, AnalogSensor := #DataIn.Orz_1_AnalSens, Standstill_Tolerance :=, Standstill_Delay := T#10MS, Filter_Tau := T#10MS, Check_AI_Value :=, Par := #Spin_Lat_1.Par, Data := #Spin_Lat_1.Data.Sens, HMI := #Spin_Lat_1.Data.HMI, Warning := #Warning.Orz_1_AnalSens, ScaleValue =>, Standstill =>)
   END_RUNG
   RUNG wire#powerrail
      Contact( #AreaInterface.Man )
   END_RUNG wire#w1
   // the same network as SCL:
   #Orz_1_AnalSens(AnalogSensor := #DataIn.Orz_1_AnalSens,   // "Analogic_SensorManagement"
                   Preset_Conditions := #AreaInterface.Man,
                   Standstill_Delay := T#10MS,
                   Filter_Tau := T#10MS,
                   Par := #Spin_Lat_1.Par,
                   Data := #Spin_Lat_1.Data.Sens,
                   HMI := #Spin_Lat_1.Data.HMI,
                   Warning := #Warning.Orz_1_AnalSens);
END_REGION

REGION Network 34: Orizzontale_1 - Allarme problemi sul sensore analogico
   RUNG wire#powerrail
      I_Contact( #Warning.Orz_1_AnalSens.PresetNeed )
      I_Contact( #Warning.Orz_1_AnalSens.SignalError )
      Not()
      wire#w1
      Contact( #CIn.Manager_SpinLat_1.Control_ON )
      wire#w2
      S_Coil( #Alarm.Orz_1_AnalSens_Issue )
   END_RUNG
   RUNG wire#w1
      Contact( #AreaInterface.Aut )
   END_RUNG wire#w2
   RUNG wire#w1
      I_Contact( #Sts.OP_CanMoveFreely )
      wire#w3
      Contact( #Orz_1.COut.Rest_CheckNext )
   END_RUNG wire#w2
   RUNG wire#w3
      Contact( #Orz_1.COut.Work_CheckNext )
   END_RUNG wire#w2
   // the same network as SCL:
   IF NOT (NOT #Warning.Orz_1_AnalSens.PresetNeed AND NOT #Warning.Orz_1_AnalSens.SignalError) AND (#CIn.Manager_SpinLat_1.Control_ON OR #AreaInterface.Aut OR (NOT #Sts.OP_CanMoveFreely AND (#Orz_1.COut.Rest_CheckNext OR #Orz_1.COut.Work_CheckNext))) THEN
       #Alarm.Orz_1_AnalSens_Issue := TRUE;
   END_IF;
END_REGION

REGION Network 35 (SCL): Orizzontale_1 - Datain / Config
   // DataIn Scritti sulla CALL dell'FB

   #Orz_1.Config := #Config.Orz_1;

   IF #Spin_Lat_1.Par.Enable AND #Sts.Beam.H_B > 0.0 THEN

       #Orz_1.DataIn.Work_Ls[1] := #Vrt_1.DataIn.Work_Ls[1] := ABS (#Orz_1_AnalSens.ScaleValue - #Sts.Beam.H_B) <= #Spin_Lat_1.Par_Mach.Tol_Work;
       #Orz_1.Config.V.WorkLimSwitchExist := TRUE;
       #Orz_1.Config.V.WorkTime := T#0.01s;

   ELSIF #Ctrl.OP_Rest THEN
       #Orz_1.DataIn.Work_Ls[1] := FALSE;
       #Vrt_1.DataIn.Work_Ls[1] := FALSE;

       // ********************************************************************************************************************************************
   ELSE
       // Overide della configurazione di default della valvola

       #Orz_1.Config.V.WorkLimSwitchExist := FALSE;
       #Orz_1.Config.V.WorkTime := #Spin_Lat_1.Par_Mach.WorkTime_SensDisable;
   END_IF;
END_REGION

REGION Network 36: Orizzontale_1 - CIn External alarm
   RUNG wire#powerrail
      I_Contact( #Alarm.Orz_1_AnalSens_Issue )
      I_Contact( #Warning.Orz_1_AnalSens.PresetNeed )
      I_Contact( #Warning.Orz_1_AnalSens.SignalError )
      Not()
      Coil( #Orz_1.Cin.ExternalAlarms )
   END_RUNG
   // the same network as SCL:
   #Orz_1.Cin.ExternalAlarms := NOT (NOT #Alarm.Orz_1_AnalSens_Issue AND NOT #Warning.Orz_1_AnalSens.PresetNeed AND NOT #Warning.Orz_1_AnalSens.SignalError);
END_REGION

REGION Network 37: Orizzontale_1 - Cin Ext Enable
   RUNG wire#powerrail
      Contact( TRUE )
      wire#w1
      Coil( #Orz_1.Cin.Rest_ExtEnable )
   END_RUNG
   RUNG wire#powerrail
      Contact( #AreaInterface.Man )
      I_Contact( #CIn.Manager_SpinLat_1.Control_ON )
      Contact( #Sts.OP_CanMoveFreely )
   END_RUNG wire#w1
   RUNG wire#powerrail
      Contact( TRUE )
      wire#w2
      Coil( #Orz_1.Cin.Work_ExtEnable )
   END_RUNG
   RUNG wire#powerrail
      Contact( #AreaInterface.Man )
      I_Contact( #CIn.Manager_SpinLat_1.Control_ON )
      Contact( #Sts.OP_CanMoveFreely )
   END_RUNG wire#w2
   // the same network as SCL:
   #Orz_1.Cin.Rest_ExtEnable := TRUE OR (#AreaInterface.Man AND NOT #CIn.Manager_SpinLat_1.Control_ON AND #Sts.OP_CanMoveFreely);
   #Orz_1.Cin.Work_ExtEnable := TRUE OR (#AreaInterface.Man AND NOT #CIn.Manager_SpinLat_1.Control_ON AND #Sts.OP_CanMoveFreely);
END_REGION

REGION Network 38: Orizzontale_1 - Valve Manager
   RUNG wire#powerrail
      #Orz_1(AreaInterface := #AreaInterface, ZSI := #ZSI, DSI := #DSI, DataIn :=, Cin :=, Config := #Config.Orz_1, Alarm := #Alarm.Orz_1, Warning := #Warning.Orz_1, MachineInterface =>, COut => #COut.Orz_1, DataOut =>)
   END_RUNG
   // the same network as SCL:
   #Orz_1(AreaInterface := #AreaInterface,   // "ValveMachine_FB"
          ZSI := #ZSI,
          DSI := #DSI,
          Config := #Config.Orz_1,
          Alarm := #Alarm.Orz_1,
          Warning := #Warning.Orz_1,
          COut => #COut.Orz_1);
END_REGION

REGION Network 39: <+>
END_REGION

REGION Network 40: Orizzontale_2 -Scalatura sensore
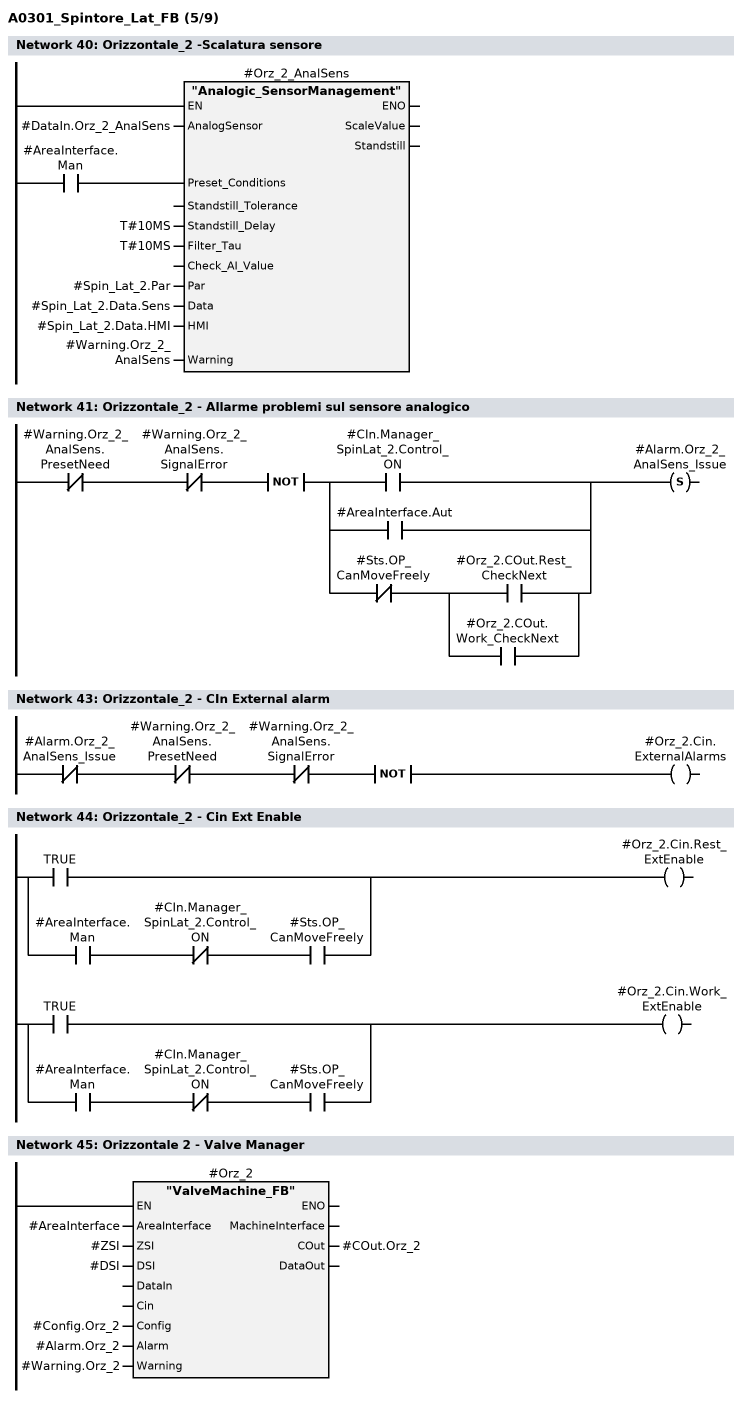
   RUNG wire#powerrail
      #Orz_2_AnalSens(Preset_Conditions := wire#w1, AnalogSensor := #DataIn.Orz_2_AnalSens, Standstill_Tolerance :=, Standstill_Delay := T#10MS, Filter_Tau := T#10MS, Check_AI_Value :=, Par := #Spin_Lat_2.Par, Data := #Spin_Lat_2.Data.Sens, HMI := #Spin_Lat_2.Data.HMI, Warning := #Warning.Orz_2_AnalSens, ScaleValue =>, Standstill =>)
   END_RUNG
   RUNG wire#powerrail
      Contact( #AreaInterface.Man )
   END_RUNG wire#w1
   // the same network as SCL:
   #Orz_2_AnalSens(AnalogSensor := #DataIn.Orz_2_AnalSens,   // "Analogic_SensorManagement"
                   Preset_Conditions := #AreaInterface.Man,
                   Standstill_Delay := T#10MS,
                   Filter_Tau := T#10MS,
                   Par := #Spin_Lat_2.Par,
                   Data := #Spin_Lat_2.Data.Sens,
                   HMI := #Spin_Lat_2.Data.HMI,
                   Warning := #Warning.Orz_2_AnalSens);
END_REGION

REGION Network 41: Orizzontale_2 - Allarme problemi sul sensore analogico
   RUNG wire#powerrail
      I_Contact( #Warning.Orz_2_AnalSens.PresetNeed )
      I_Contact( #Warning.Orz_2_AnalSens.SignalError )
      Not()
      wire#w1
      Contact( #CIn.Manager_SpinLat_2.Control_ON )
      wire#w2
      S_Coil( #Alarm.Orz_2_AnalSens_Issue )
   END_RUNG
   RUNG wire#w1
      Contact( #AreaInterface.Aut )
   END_RUNG wire#w2
   RUNG wire#w1
      I_Contact( #Sts.OP_CanMoveFreely )
      wire#w3
      Contact( #Orz_2.COut.Rest_CheckNext )
   END_RUNG wire#w2
   RUNG wire#w3
      Contact( #Orz_2.COut.Work_CheckNext )
   END_RUNG wire#w2
   // the same network as SCL:
   IF NOT (NOT #Warning.Orz_2_AnalSens.PresetNeed AND NOT #Warning.Orz_2_AnalSens.SignalError) AND (#CIn.Manager_SpinLat_2.Control_ON OR #AreaInterface.Aut OR (NOT #Sts.OP_CanMoveFreely AND (#Orz_2.COut.Rest_CheckNext OR #Orz_2.COut.Work_CheckNext))) THEN
       #Alarm.Orz_2_AnalSens_Issue := TRUE;
   END_IF;
END_REGION

REGION Network 42 (SCL): Orizzontale_2 - Datain / Config
   // DataIn Scritti sulla CALL dell'FB
   #Orz_2.Config := #Config.Orz_2;
   #Spin_Lat_2.Par.Enable := TRUE;

   // Se dal controllo di misura la lunghezza del Beam supera la Quota di abilitazione Spintore 2 abilito il controllo del sensore compensatore sul cilindro ORZ
   IF #Sts."En/Dis_SpinLat_2" THEN

   // *******************************************************************************************************************
   IF  #Spin_Lat_2.Par.Enable AND #Sts.Beam.H_B > 0.0 THEN
       #Spin_Lat_2.Par_Mach.Tol_Work := #Spin_Lat_1.Par_Mach.Tol_Work;

       #Orz_2.DataIn.Work_Ls[1] := #Vrt_2.DataIn.Work_Ls[1] := ABS (#Orz_2_AnalSens.ScaleValue - #Sts.Beam.H_B) <= #Spin_Lat_2.Par_Mach.Tol_Work;
       #Orz_2.Config.V.WorkLimSwitchExist := TRUE;
       #Orz_2.Config.V.WorkTime := T#0.01s;

   ELSIF #Ctrl.OP_Rest THEN
       #Orz_2.DataIn.Work_Ls[1] := FALSE;
       #Vrt_2.DataIn.Work_Ls[1] := FALSE;

       // ***************************************************************************************************************
   ELSE
       // Overide della configurazione di default della valvola

       #Orz_2.DataIn.Work_Ls[1] := FALSE;
       #Orz_2.Config.V.WorkLimSwitchExist := FALSE;
       #Orz_2.Config.V.WorkTime := #Spin_Lat_2.Par_Mach.WorkTime_SensDisable;
   END_IF;
   END_IF;
END_REGION

REGION Network 43: Orizzontale_2 - CIn External alarm
   RUNG wire#powerrail
      I_Contact( #Alarm.Orz_2_AnalSens_Issue )
      I_Contact( #Warning.Orz_2_AnalSens.PresetNeed )
      I_Contact( #Warning.Orz_2_AnalSens.SignalError )
      Not()
      Coil( #Orz_2.Cin.ExternalAlarms )
   END_RUNG
   // the same network as SCL:
   #Orz_2.Cin.ExternalAlarms := NOT (NOT #Alarm.Orz_2_AnalSens_Issue AND NOT #Warning.Orz_2_AnalSens.PresetNeed AND NOT #Warning.Orz_2_AnalSens.SignalError);
END_REGION

REGION Network 44: Orizzontale_2 - Cin Ext Enable
   RUNG wire#powerrail
      Contact( TRUE )
      wire#w1
      Coil( #Orz_2.Cin.Rest_ExtEnable )
   END_RUNG
   RUNG wire#powerrail
      Contact( #AreaInterface.Man )
      I_Contact( #CIn.Manager_SpinLat_2.Control_ON )
      Contact( #Sts.OP_CanMoveFreely )
   END_RUNG wire#w1
   RUNG wire#powerrail
      Contact( TRUE )
      wire#w2
      Coil( #Orz_2.Cin.Work_ExtEnable )
   END_RUNG
   RUNG wire#powerrail
      Contact( #AreaInterface.Man )
      I_Contact( #CIn.Manager_SpinLat_2.Control_ON )
      Contact( #Sts.OP_CanMoveFreely )
   END_RUNG wire#w2
   // the same network as SCL:
   #Orz_2.Cin.Rest_ExtEnable := TRUE OR (#AreaInterface.Man AND NOT #CIn.Manager_SpinLat_2.Control_ON AND #Sts.OP_CanMoveFreely);
   #Orz_2.Cin.Work_ExtEnable := TRUE OR (#AreaInterface.Man AND NOT #CIn.Manager_SpinLat_2.Control_ON AND #Sts.OP_CanMoveFreely);
END_REGION

REGION Network 45: Orizzontale 2 - Valve Manager
   RUNG wire#powerrail
      #Orz_2(AreaInterface := #AreaInterface, ZSI := #ZSI, DSI := #DSI, DataIn :=, Cin :=, Config := #Config.Orz_2, Alarm := #Alarm.Orz_2, Warning := #Warning.Orz_2, MachineInterface =>, COut => #COut.Orz_2, DataOut =>)
   END_RUNG
   // the same network as SCL:
   #Orz_2(AreaInterface := #AreaInterface,   // "ValveMachine_FB"
          ZSI := #ZSI,
          DSI := #DSI,
          Config := #Config.Orz_2,
          Alarm := #Alarm.Orz_2,
          Warning := #Warning.Orz_2,
          COut => #COut.Orz_2);
END_REGION

REGION Network 47: << GESTIONE SOLLEVATORI >>
END_REGION

REGION Network 48: S[1...6] Sollevatori - CIn External alarm
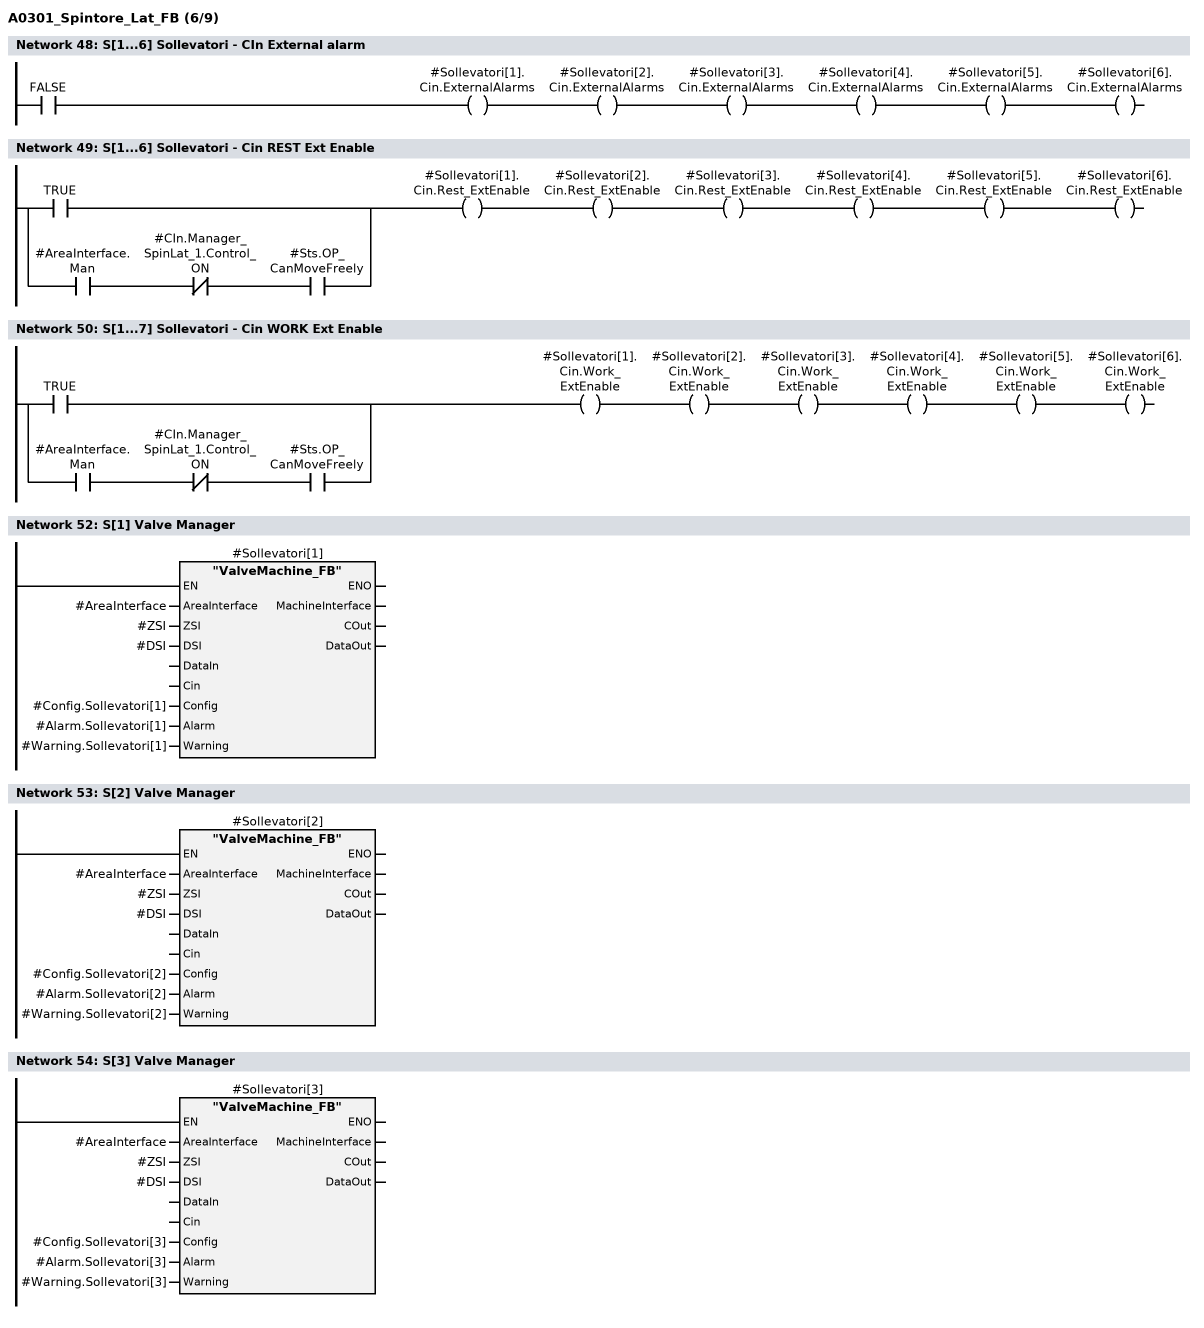
   RUNG wire#powerrail
      Contact( FALSE )
      Coil( #Sollevatori[1].Cin.ExternalAlarms )
      Coil( #Sollevatori[2].Cin.ExternalAlarms )
      Coil( #Sollevatori[3].Cin.ExternalAlarms )
      Coil( #Sollevatori[4].Cin.ExternalAlarms )
      Coil( #Sollevatori[5].Cin.ExternalAlarms )
      Coil( #Sollevatori[6].Cin.ExternalAlarms )
   END_RUNG
   // the same network as SCL:
   #Sollevatori[1].Cin.ExternalAlarms := FALSE;
   #Sollevatori[2].Cin.ExternalAlarms := FALSE;
   #Sollevatori[3].Cin.ExternalAlarms := FALSE;
   #Sollevatori[4].Cin.ExternalAlarms := FALSE;
   #Sollevatori[5].Cin.ExternalAlarms := FALSE;
   #Sollevatori[6].Cin.ExternalAlarms := FALSE;
END_REGION

REGION Network 49: S[1...6] Sollevatori - Cin REST Ext Enable
   RUNG wire#powerrail
      Contact( TRUE )
      wire#w1
      Coil( #Sollevatori[1].Cin.Rest_ExtEnable )
      Coil( #Sollevatori[2].Cin.Rest_ExtEnable )
      Coil( #Sollevatori[3].Cin.Rest_ExtEnable )
      Coil( #Sollevatori[4].Cin.Rest_ExtEnable )
      Coil( #Sollevatori[5].Cin.Rest_ExtEnable )
      Coil( #Sollevatori[6].Cin.Rest_ExtEnable )
   END_RUNG
   RUNG wire#powerrail
      Contact( #AreaInterface.Man )
      I_Contact( #CIn.Manager_SpinLat_1.Control_ON )
      Contact( #Sts.OP_CanMoveFreely )
   END_RUNG wire#w1
   // the same network as SCL:
   #Sollevatori[1].Cin.Rest_ExtEnable := TRUE OR (#AreaInterface.Man AND NOT #CIn.Manager_SpinLat_1.Control_ON AND #Sts.OP_CanMoveFreely);
   #Sollevatori[2].Cin.Rest_ExtEnable := TRUE OR (#AreaInterface.Man AND NOT #CIn.Manager_SpinLat_1.Control_ON AND #Sts.OP_CanMoveFreely);
   #Sollevatori[3].Cin.Rest_ExtEnable := TRUE OR (#AreaInterface.Man AND NOT #CIn.Manager_SpinLat_1.Control_ON AND #Sts.OP_CanMoveFreely);
   #Sollevatori[4].Cin.Rest_ExtEnable := TRUE OR (#AreaInterface.Man AND NOT #CIn.Manager_SpinLat_1.Control_ON AND #Sts.OP_CanMoveFreely);
   #Sollevatori[5].Cin.Rest_ExtEnable := TRUE OR (#AreaInterface.Man AND NOT #CIn.Manager_SpinLat_1.Control_ON AND #Sts.OP_CanMoveFreely);
   #Sollevatori[6].Cin.Rest_ExtEnable := TRUE OR (#AreaInterface.Man AND NOT #CIn.Manager_SpinLat_1.Control_ON AND #Sts.OP_CanMoveFreely);
END_REGION

REGION Network 50: S[1...7] Sollevatori - Cin WORK Ext Enable
   RUNG wire#powerrail
      Contact( TRUE )
      wire#w1
      Coil( #Sollevatori[1].Cin.Work_ExtEnable )
      Coil( #Sollevatori[2].Cin.Work_ExtEnable )
      Coil( #Sollevatori[3].Cin.Work_ExtEnable )
      Coil( #Sollevatori[4].Cin.Work_ExtEnable )
      Coil( #Sollevatori[5].Cin.Work_ExtEnable )
      Coil( #Sollevatori[6].Cin.Work_ExtEnable )
   END_RUNG
   RUNG wire#powerrail
      Contact( #AreaInterface.Man )
      I_Contact( #CIn.Manager_SpinLat_1.Control_ON )
      Contact( #Sts.OP_CanMoveFreely )
   END_RUNG wire#w1
   // the same network as SCL:
   #Sollevatori[1].Cin.Work_ExtEnable := TRUE OR (#AreaInterface.Man AND NOT #CIn.Manager_SpinLat_1.Control_ON AND #Sts.OP_CanMoveFreely);
   #Sollevatori[2].Cin.Work_ExtEnable := TRUE OR (#AreaInterface.Man AND NOT #CIn.Manager_SpinLat_1.Control_ON AND #Sts.OP_CanMoveFreely);
   #Sollevatori[3].Cin.Work_ExtEnable := TRUE OR (#AreaInterface.Man AND NOT #CIn.Manager_SpinLat_1.Control_ON AND #Sts.OP_CanMoveFreely);
   #Sollevatori[4].Cin.Work_ExtEnable := TRUE OR (#AreaInterface.Man AND NOT #CIn.Manager_SpinLat_1.Control_ON AND #Sts.OP_CanMoveFreely);
   #Sollevatori[5].Cin.Work_ExtEnable := TRUE OR (#AreaInterface.Man AND NOT #CIn.Manager_SpinLat_1.Control_ON AND #Sts.OP_CanMoveFreely);
   #Sollevatori[6].Cin.Work_ExtEnable := TRUE OR (#AreaInterface.Man AND NOT #CIn.Manager_SpinLat_1.Control_ON AND #Sts.OP_CanMoveFreely);
END_REGION

REGION Network 51: <+>
END_REGION

REGION Network 52: S[1] Valve Manager
   RUNG wire#powerrail
      #Sollevatori[1](AreaInterface := #AreaInterface, ZSI := #ZSI, DSI := #DSI, DataIn :=, Cin :=, Config := #Config.Sollevatori[1], Alarm := #Alarm.Sollevatori[1], Warning := #Warning.Sollevatori[1], MachineInterface =>, COut =>, DataOut =>)
   END_RUNG
   // the same network as SCL:
   #Sollevatori[1](AreaInterface := #AreaInterface,   // "ValveMachine_FB"
                   ZSI := #ZSI,
                   DSI := #DSI,
                   Config := #Config.Sollevatori[1],
                   Alarm := #Alarm.Sollevatori[1],
                   Warning := #Warning.Sollevatori[1]);
END_REGION

REGION Network 53: S[2] Valve Manager
   RUNG wire#powerrail
      #Sollevatori[2](AreaInterface := #AreaInterface, ZSI := #ZSI, DSI := #DSI, DataIn :=, Cin :=, Config := #Config.Sollevatori[2], Alarm := #Alarm.Sollevatori[2], Warning := #Warning.Sollevatori[2], MachineInterface =>, COut =>, DataOut =>)
   END_RUNG
   // the same network as SCL:
   #Sollevatori[2](AreaInterface := #AreaInterface,   // "ValveMachine_FB"
                   ZSI := #ZSI,
                   DSI := #DSI,
                   Config := #Config.Sollevatori[2],
                   Alarm := #Alarm.Sollevatori[2],
                   Warning := #Warning.Sollevatori[2]);
END_REGION

REGION Network 54: S[3] Valve Manager
   RUNG wire#powerrail
      #Sollevatori[3](AreaInterface := #AreaInterface, ZSI := #ZSI, DSI := #DSI, DataIn :=, Cin :=, Config := #Config.Sollevatori[3], Alarm := #Alarm.Sollevatori[3], Warning := #Warning.Sollevatori[3], MachineInterface =>, COut =>, DataOut =>)
   END_RUNG
   // the same network as SCL:
   #Sollevatori[3](AreaInterface := #AreaInterface,   // "ValveMachine_FB"
                   ZSI := #ZSI,
                   DSI := #DSI,
                   Config := #Config.Sollevatori[3],
                   Alarm := #Alarm.Sollevatori[3],
                   Warning := #Warning.Sollevatori[3]);
END_REGION

REGION Network 55: S[4] Valve Manager
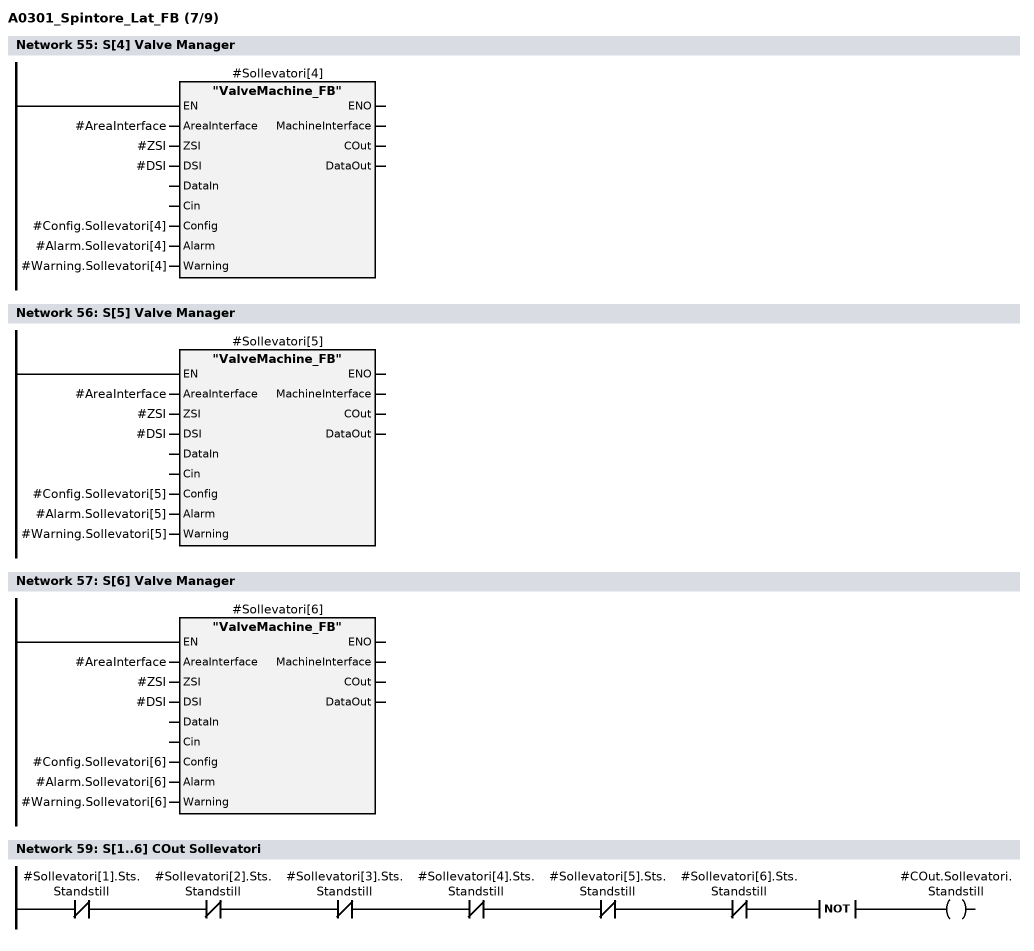
   RUNG wire#powerrail
      #Sollevatori[4](AreaInterface := #AreaInterface, ZSI := #ZSI, DSI := #DSI, DataIn :=, Cin :=, Config := #Config.Sollevatori[4], Alarm := #Alarm.Sollevatori[4], Warning := #Warning.Sollevatori[4], MachineInterface =>, COut =>, DataOut =>)
   END_RUNG
   // the same network as SCL:
   #Sollevatori[4](AreaInterface := #AreaInterface,   // "ValveMachine_FB"
                   ZSI := #ZSI,
                   DSI := #DSI,
                   Config := #Config.Sollevatori[4],
                   Alarm := #Alarm.Sollevatori[4],
                   Warning := #Warning.Sollevatori[4]);
END_REGION

REGION Network 56: S[5] Valve Manager
   RUNG wire#powerrail
      #Sollevatori[5](AreaInterface := #AreaInterface, ZSI := #ZSI, DSI := #DSI, DataIn :=, Cin :=, Config := #Config.Sollevatori[5], Alarm := #Alarm.Sollevatori[5], Warning := #Warning.Sollevatori[5], MachineInterface =>, COut =>, DataOut =>)
   END_RUNG
   // the same network as SCL:
   #Sollevatori[5](AreaInterface := #AreaInterface,   // "ValveMachine_FB"
                   ZSI := #ZSI,
                   DSI := #DSI,
                   Config := #Config.Sollevatori[5],
                   Alarm := #Alarm.Sollevatori[5],
                   Warning := #Warning.Sollevatori[5]);
END_REGION

REGION Network 57: S[6] Valve Manager
   RUNG wire#powerrail
      #Sollevatori[6](AreaInterface := #AreaInterface, ZSI := #ZSI, DSI := #DSI, DataIn :=, Cin :=, Config := #Config.Sollevatori[6], Alarm := #Alarm.Sollevatori[6], Warning := #Warning.Sollevatori[6], MachineInterface =>, COut =>, DataOut =>)
   END_RUNG
   // the same network as SCL:
   #Sollevatori[6](AreaInterface := #AreaInterface,   // "ValveMachine_FB"
                   ZSI := #ZSI,
                   DSI := #DSI,
                   Config := #Config.Sollevatori[6],
                   Alarm := #Alarm.Sollevatori[6],
                   Warning := #Warning.Sollevatori[6]);
END_REGION

REGION Network 58: <+>
END_REGION

REGION Network 59: S[1..6] COut Sollevatori
   RUNG wire#powerrail
      I_Contact( #Sollevatori[1].Sts.Standstill )
      I_Contact( #Sollevatori[2].Sts.Standstill )
      I_Contact( #Sollevatori[3].Sts.Standstill )
      I_Contact( #Sollevatori[4].Sts.Standstill )
      I_Contact( #Sollevatori[5].Sts.Standstill )
      I_Contact( #Sollevatori[6].Sts.Standstill )
      Not()
      Coil( #COut.Sollevatori.Standstill )
   END_RUNG
   // the same network as SCL:
   #COut.Sollevatori.Standstill := NOT (NOT #Sollevatori[1].Sts.Standstill AND NOT #Sollevatori[2].Sts.Standstill AND NOT #Sollevatori[3].Sts.Standstill AND NOT #Sollevatori[4].Sts.Standstill AND NOT #Sollevatori[5].Sts.Standstill AND NOT #Sollevatori[6].Sts.Standstill);
END_REGION

REGION Network 60 (SCL): S[1..6] COut Sollevatori


   // Controllo uscita COut AT_REST in base allo stato di tutti i Sollevatori
   IF  #Sollevatori[1].COut.Rest AND
       #Sollevatori[2].COut.Rest AND
       #Sollevatori[3].COut.Rest AND
       #Sollevatori[4].COut.Rest AND
       #Sollevatori[5].COut.Rest AND
       #Sollevatori[6].COut.Rest THEN
       #COut.Sollevatori.Rest := 1;
   ELSE
       #COut.Sollevatori.Rest := 0;
   END_IF;

   // Controllo uscita COut AT_WORK in base allo stato di tutti i Sollevatori
   IF  #Sollevatori[1].COut.Work AND
       #Sollevatori[2].COut.Work AND
       #Sollevatori[3].COut.Work AND
       #Sollevatori[4].COut.Work AND
       #Sollevatori[5].COut.Work AND
       #Sollevatori[6].COut.Work THEN
       #COut.Sollevatori.Work := 1;
   ELSE
       #COut.Sollevatori.Work := 0;
   END_IF;
END_REGION

REGION Network 61: <+>
END_REGION

REGION Network 62: Stazione COut
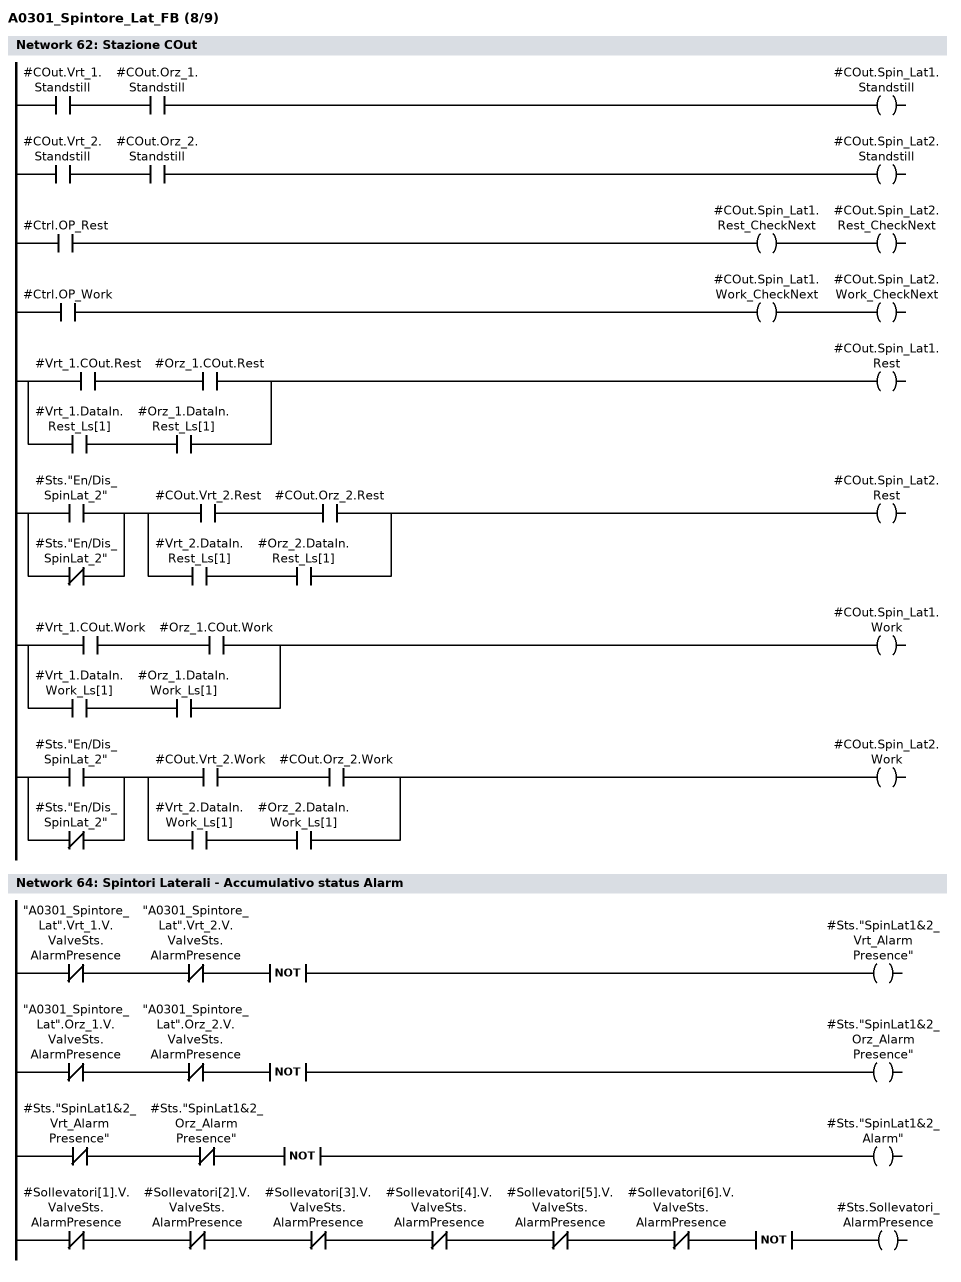
   RUNG wire#powerrail
      Contact( #COut.Vrt_1.Standstill )
      Contact( #COut.Orz_1.Standstill )
      Coil( #COut.Spin_Lat1.Standstill )
   END_RUNG
   RUNG wire#powerrail
      Contact( #COut.Vrt_2.Standstill )
      Contact( #COut.Orz_2.Standstill )
      Coil( #COut.Spin_Lat2.Standstill )
   END_RUNG
   RUNG wire#powerrail
      Contact( #Ctrl.OP_Rest )
      Coil( #COut.Spin_Lat1.Rest_CheckNext )
      Coil( #COut.Spin_Lat2.Rest_CheckNext )
   END_RUNG
   RUNG wire#powerrail
      Contact( #Ctrl.OP_Work )
      Coil( #COut.Spin_Lat1.Work_CheckNext )
      Coil( #COut.Spin_Lat2.Work_CheckNext )
   END_RUNG
   RUNG wire#powerrail
      Contact( #Vrt_1.COut.Rest )
      Contact( #Orz_1.COut.Rest )
      wire#w1
      Coil( #COut.Spin_Lat1.Rest )
   END_RUNG
   RUNG wire#powerrail
      Contact( #Vrt_1.DataIn.Rest_Ls[1] )
      Contact( #Orz_1.DataIn.Rest_Ls[1] )
   END_RUNG wire#w1
   RUNG wire#powerrail
      Contact( #Sts."En/Dis_SpinLat_2" )
      wire#w2
      Contact( #COut.Vrt_2.Rest )
      Contact( #COut.Orz_2.Rest )
      wire#w3
      Coil( #COut.Spin_Lat2.Rest )
   END_RUNG
   RUNG wire#powerrail
      I_Contact( #Sts."En/Dis_SpinLat_2" )
   END_RUNG wire#w2
   RUNG wire#w2
      Contact( #Vrt_2.DataIn.Rest_Ls[1] )
      Contact( #Orz_2.DataIn.Rest_Ls[1] )
   END_RUNG wire#w3
   RUNG wire#powerrail
      Contact( #Vrt_1.COut.Work )
      Contact( #Orz_1.COut.Work )
      wire#w4
      Coil( #COut.Spin_Lat1.Work )
   END_RUNG
   RUNG wire#powerrail
      Contact( #Vrt_1.DataIn.Work_Ls[1] )
      Contact( #Orz_1.DataIn.Work_Ls[1] )
   END_RUNG wire#w4
   RUNG wire#powerrail
      Contact( #Sts."En/Dis_SpinLat_2" )
      wire#w5
      Contact( #COut.Vrt_2.Work )
      Contact( #COut.Orz_2.Work )
      wire#w6
      Coil( #COut.Spin_Lat2.Work )
   END_RUNG
   RUNG wire#powerrail
      I_Contact( #Sts."En/Dis_SpinLat_2" )
   END_RUNG wire#w5
   RUNG wire#w5
      Contact( #Vrt_2.DataIn.Work_Ls[1] )
      Contact( #Orz_2.DataIn.Work_Ls[1] )
   END_RUNG wire#w6
   // the same network as SCL:
   #COut.Spin_Lat1.Standstill := #COut.Vrt_1.Standstill AND #COut.Orz_1.Standstill;
   #COut.Spin_Lat2.Standstill := #COut.Vrt_2.Standstill AND #COut.Orz_2.Standstill;
   #COut.Spin_Lat1.Rest_CheckNext := #Ctrl.OP_Rest;
   #COut.Spin_Lat2.Rest_CheckNext := #Ctrl.OP_Rest;
   #COut.Spin_Lat1.Work_CheckNext := #Ctrl.OP_Work;
   #COut.Spin_Lat2.Work_CheckNext := #Ctrl.OP_Work;
   #COut.Spin_Lat1.Rest := (#Vrt_1.COut.Rest AND #Orz_1.COut.Rest) OR (#Vrt_1.DataIn.Rest_Ls[1] AND #Orz_1.DataIn.Rest_Ls[1]);
   #COut.Spin_Lat2.Rest := (#Sts."En/Dis_SpinLat_2" OR NOT #Sts."En/Dis_SpinLat_2") AND ((#COut.Vrt_2.Rest AND #COut.Orz_2.Rest) OR (#Vrt_2.DataIn.Rest_Ls[1] AND #Orz_2.DataIn.Rest_Ls[1]));
   #COut.Spin_Lat1.Work := (#Vrt_1.COut.Work AND #Orz_1.COut.Work) OR (#Vrt_1.DataIn.Work_Ls[1] AND #Orz_1.DataIn.Work_Ls[1]);
   #COut.Spin_Lat2.Work := (#Sts."En/Dis_SpinLat_2" OR NOT #Sts."En/Dis_SpinLat_2") AND ((#COut.Vrt_2.Work AND #COut.Orz_2.Work) OR (#Vrt_2.DataIn.Work_Ls[1] AND #Orz_2.DataIn.Work_Ls[1]));
END_REGION

REGION Network 64: Spintori Laterali - Accumulativo status Alarm
   RUNG wire#powerrail
      I_Contact( "A0301_Spintore_Lat".Vrt_1.V.ValveSts.AlarmPresence )
      I_Contact( "A0301_Spintore_Lat".Vrt_2.V.ValveSts.AlarmPresence )
      Not()
      Coil( #Sts."SpinLat1&2_Vrt_AlarmPresence" )
   END_RUNG
   RUNG wire#powerrail
      I_Contact( "A0301_Spintore_Lat".Orz_1.V.ValveSts.AlarmPresence )
      I_Contact( "A0301_Spintore_Lat".Orz_2.V.ValveSts.AlarmPresence )
      Not()
      Coil( #Sts."SpinLat1&2_Orz_AlarmPresence" )
   END_RUNG
   RUNG wire#powerrail
      I_Contact( #Sts."SpinLat1&2_Vrt_AlarmPresence" )
      I_Contact( #Sts."SpinLat1&2_Orz_AlarmPresence" )
      Not()
      Coil( #Sts."SpinLat1&2_Alarm" )
   END_RUNG
   RUNG wire#powerrail
      I_Contact( #Sollevatori[1].V.ValveSts.AlarmPresence )
      I_Contact( #Sollevatori[2].V.ValveSts.AlarmPresence )
      I_Contact( #Sollevatori[3].V.ValveSts.AlarmPresence )
      I_Contact( #Sollevatori[4].V.ValveSts.AlarmPresence )
      I_Contact( #Sollevatori[5].V.ValveSts.AlarmPresence )
      I_Contact( #Sollevatori[6].V.ValveSts.AlarmPresence )
      Not()
      Coil( #Sts.Sollevatori_AlarmPresence )
   END_RUNG
   // the same network as SCL:
   #Sts."SpinLat1&2_Vrt_AlarmPresence" := NOT (NOT "A0301_Spintore_Lat".Vrt_1.V.ValveSts.AlarmPresence AND NOT "A0301_Spintore_Lat".Vrt_2.V.ValveSts.AlarmPresence);
   #Sts."SpinLat1&2_Orz_AlarmPresence" := NOT (NOT "A0301_Spintore_Lat".Orz_1.V.ValveSts.AlarmPresence AND NOT "A0301_Spintore_Lat".Orz_2.V.ValveSts.AlarmPresence);
   #Sts."SpinLat1&2_Alarm" := NOT (NOT #Sts."SpinLat1&2_Vrt_AlarmPresence" AND NOT #Sts."SpinLat1&2_Orz_AlarmPresence");
   #Sts.Sollevatori_AlarmPresence := NOT (NOT #Sollevatori[1].V.ValveSts.AlarmPresence AND NOT #Sollevatori[2].V.ValveSts.AlarmPresence AND NOT #Sollevatori[3].V.ValveSts.AlarmPresence AND NOT #Sollevatori[4].V.ValveSts.AlarmPresence AND NOT #Sollevatori[5].V.ValveSts.AlarmPresence AND NOT #Sollevatori[6].V.ValveSts.AlarmPresence);
END_REGION

REGION Network 65 (SCL): HMI STATUS - Postazione
   // Area dati appoggio per HMI
   // SPINTORE LAT. 1&2 Verticale
   #HMI."SpinLat1&2_Vrt_Sts".Standstill := #COut.Vrt_1.Standstill AND #COut.Vrt_2.Standstill;
   #HMI."SpinLat1&2_Vrt_Sts".Rest := #COut.Vrt_1.Rest AND (#COut.Vrt_2.Rest OR NOT #Sts."En/Dis_SpinLat_2");
   #HMI."SpinLat1&2_Vrt_Sts".Work := #COut.Vrt_1.Work AND (#COut.Vrt_2.Work OR NOT #Sts."En/Dis_SpinLat_2");
   #HMI."SpinLat1&2_Vrt_Sts".AlarmPresence := #Sts."SpinLat1&2_Vrt_AlarmPresence";

   // SPINTORE LAT. 1&2 Orizzontale
   #HMI."SpinLat1&2_Orz_Sts".Standstill := #COut.Orz_1.Standstill AND #COut.Orz_2.Standstill;
   #HMI."SpinLat1&2_Orz_Sts".Rest := #COut.Orz_1.Rest AND (#COut.Orz_2.Rest OR NOT #Sts."En/Dis_SpinLat_2");
   #HMI."SpinLat1&2_Orz_Sts".Work := #COut.Orz_1.Work AND (#COut.Orz_2.Work OR NOT #Sts."En/Dis_SpinLat_2");
   #HMI."SpinLat1&2_Orz_Sts".AlarmPresence := #Sts."SpinLat1&2_Orz_AlarmPresence";

   // Stazione spintori laterati
   #HMI."SpinLat1&2_Sts".Standstill := #COut.Spin_Lat1.Standstill AND (#COut.Spin_Lat2.Standstill OR NOT #Sts."En/Dis_SpinLat_2");
   #HMI."SpinLat1&2_Sts".Rest := #COut.Spin_Lat1.Rest AND (#COut.Spin_Lat2.Rest OR NOT #Sts."En/Dis_SpinLat_2");
   #HMI."SpinLat1&2_Sts".Work := #COut.Spin_Lat1.Work AND(#COut.Spin_Lat2.Work OR NOT #Sts."En/Dis_SpinLat_2");
   #HMI."SpinLat1&2_Sts".AlarmPresence := #Sts."SpinLat1&2_Alarm";

   // Sollevatori
   #HMI.Sollevatori_Sts.Standstill := #COut.Sollevatori.Standstill;
   #HMI.Sollevatori_Sts.Rest := #COut.Sollevatori.Rest;
   #HMI.Sollevatori_Sts.Work := #COut.Sollevatori.Work;
   #HMI.Sollevatori_Sts.AlarmPresence := #Sts.Sollevatori_AlarmPresence;
END_REGION

REGION Network 67: << MAIN MACHINE STATUS >>
END_REGION

REGION Network 68: Machine interface
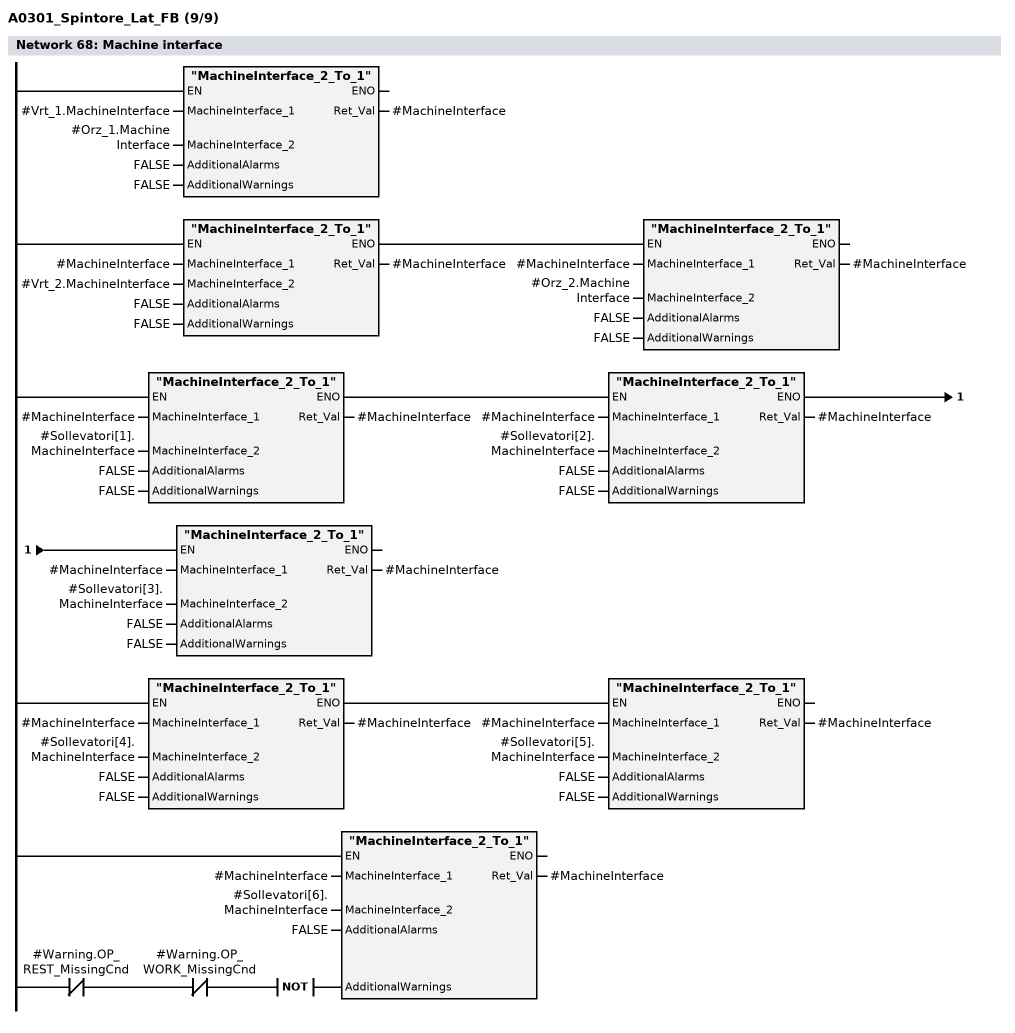
   RUNG wire#powerrail
      "MachineInterface_2_To_1"(MachineInterface_1 := #Vrt_1.MachineInterface, MachineInterface_2 := #Orz_1.MachineInterface, AdditionalAlarms := FALSE, AdditionalWarnings := FALSE, Ret_Val => #MachineInterface)
   END_RUNG
   RUNG wire#powerrail
      "MachineInterface_2_To_1"(MachineInterface_1 := #MachineInterface, MachineInterface_2 := #Vrt_2.MachineInterface, AdditionalAlarms := FALSE, AdditionalWarnings := FALSE, Ret_Val => #MachineInterface)
      "MachineInterface_2_To_1"(MachineInterface_1 := #MachineInterface, MachineInterface_2 := #Orz_2.MachineInterface, AdditionalAlarms := FALSE, AdditionalWarnings := FALSE, Ret_Val => #MachineInterface)
   END_RUNG
   RUNG wire#powerrail
      "MachineInterface_2_To_1"(MachineInterface_1 := #MachineInterface, MachineInterface_2 := #Sollevatori[1].MachineInterface, AdditionalAlarms := FALSE, AdditionalWarnings := FALSE, Ret_Val => #MachineInterface)
      "MachineInterface_2_To_1"(MachineInterface_1 := #MachineInterface, MachineInterface_2 := #Sollevatori[2].MachineInterface, AdditionalAlarms := FALSE, AdditionalWarnings := FALSE, Ret_Val => #MachineInterface)
      "MachineInterface_2_To_1"(MachineInterface_1 := #MachineInterface, MachineInterface_2 := #Sollevatori[3].MachineInterface, AdditionalAlarms := FALSE, AdditionalWarnings := FALSE, Ret_Val => #MachineInterface)
   END_RUNG
   RUNG wire#powerrail
      "MachineInterface_2_To_1"(MachineInterface_1 := #MachineInterface, MachineInterface_2 := #Sollevatori[4].MachineInterface, AdditionalAlarms := FALSE, AdditionalWarnings := FALSE, Ret_Val => #MachineInterface)
      "MachineInterface_2_To_1"(MachineInterface_1 := #MachineInterface, MachineInterface_2 := #Sollevatori[5].MachineInterface, AdditionalAlarms := FALSE, AdditionalWarnings := FALSE, Ret_Val => #MachineInterface)
   END_RUNG
   RUNG wire#powerrail
      "MachineInterface_2_To_1"(AdditionalWarnings := wire#w1, MachineInterface_1 := #MachineInterface, MachineInterface_2 := #Sollevatori[6].MachineInterface, AdditionalAlarms := FALSE, Ret_Val => #MachineInterface)
   END_RUNG
   RUNG wire#powerrail
      I_Contact( #Warning.OP_REST_MissingCnd )
      I_Contact( #Warning.OP_WORK_MissingCnd )
      Not()
   END_RUNG wire#w1
   // the same network as SCL:
   #MachineInterface := "MachineInterface_2_To_1"(MachineInterface_1 := #Vrt_1.MachineInterface,
                           MachineInterface_2 := #Orz_1.MachineInterface,
                           AdditionalAlarms := FALSE,
                           AdditionalWarnings := FALSE);
   #MachineInterface := "MachineInterface_2_To_1"(MachineInterface_1 := #MachineInterface,
                           MachineInterface_2 := #Vrt_2.MachineInterface,
                           AdditionalAlarms := FALSE,
                           AdditionalWarnings := FALSE,
                           ENO => #_w1);
   IF #_w1 THEN
       #MachineInterface := "MachineInterface_2_To_1"(MachineInterface_1 := #MachineInterface,
                               MachineInterface_2 := #Orz_2.MachineInterface,
                               AdditionalAlarms := FALSE,
                               AdditionalWarnings := FALSE);
   END_IF;
   #MachineInterface := "MachineInterface_2_To_1"(MachineInterface_1 := #MachineInterface,
                           MachineInterface_2 := #Sollevatori[1].MachineInterface,
                           AdditionalAlarms := FALSE,
                           AdditionalWarnings := FALSE,
                           ENO => #_w2);
   #MachineInterface := "MachineInterface_2_To_1"(EN := #_w2,
                           MachineInterface_1 := #MachineInterface,
                           MachineInterface_2 := #Sollevatori[2].MachineInterface,
                           AdditionalAlarms := FALSE,
                           AdditionalWarnings := FALSE,
                           ENO => #_w3);
   IF #_w3 THEN
       #MachineInterface := "MachineInterface_2_To_1"(MachineInterface_1 := #MachineInterface,
                               MachineInterface_2 := #Sollevatori[3].MachineInterface,
                               AdditionalAlarms := FALSE,
                               AdditionalWarnings := FALSE);
   END_IF;
   #MachineInterface := "MachineInterface_2_To_1"(MachineInterface_1 := #MachineInterface,
                           MachineInterface_2 := #Sollevatori[4].MachineInterface,
                           AdditionalAlarms := FALSE,
                           AdditionalWarnings := FALSE,
                           ENO => #_w4);
   IF #_w4 THEN
       #MachineInterface := "MachineInterface_2_To_1"(MachineInterface_1 := #MachineInterface,
                               MachineInterface_2 := #Sollevatori[5].MachineInterface,
                               AdditionalAlarms := FALSE,
                               AdditionalWarnings := FALSE);
   END_IF;
   #MachineInterface := "MachineInterface_2_To_1"(MachineInterface_1 := #MachineInterface,
                           MachineInterface_2 := #Sollevatori[6].MachineInterface,
                           AdditionalAlarms := FALSE,
                           AdditionalWarnings := NOT (NOT #Warning.OP_REST_MissingCnd AND NOT #Warning.OP_WORK_MissingCnd));
END_REGION
END_FUNCTION_BLOCK

FUNCTION "A0302_Manager_CALL" : Void   // FC180, LAD
// stored: SetENOAutomatically false
BEGIN

REGION Network 2 (SCL): << TRASFERIMENTO stati CIn del blocco >>
   // TRASFERIMENTO CIn UTENZE FERMI P5

   "A0302_Manager".CIn.P5.Sollevatori := "A0301_Spintore_Lat".COut.Sollevatori;
   "A0302_Manager".CIn.P5.Spintore_Lat.Spin_Lat1 := "A0301_Spintore_Lat".COut.Spin_Lat1;
   "A0302_Manager".CIn.P5.Spintore_Lat.Spin_Lat2 := "A0301_Spintore_Lat".COut.Spin_Lat2;

   "A0302_Manager".CIn.P5.SpintoreLong.Ax := "A0302_Spintore".COut.Ax;
   "A0302_Manager".CIn.P5.SpintoreLong.Ax_Sts := "A0302_Spintore".COut.Ax_Sts;
   "A0302_Manager".CIn.P5.SpintoreLong.Spintore := "A0302_Spintore".COut.Spintore;
   "A0302_Manager".CIn.P5.SpintoreLong.Vrt := "A0302_Spintore".COut.Vrt;
   "A0302_Manager".CIn.P5.SpintoreLong.Orz := "A0302_Spintore".COut.Orz;
   "A0302_Manager".CIn.P5.SpintoreLong.Sens.FTC_FuoriIngombro := "A0302_Spintore".IEC.FTC_On;

   // TRASFERIMENTO CIn BORDATRICE
   "A0302_Manager".CIn.Bordatrice.Ax := "A0302_Bordatrice".COut.Ax;
   "A0302_Manager".CIn.Bordatrice.Sts := "A0302_Bordatrice".COut.Sts;
   "A0302_Manager".CIn.Bordatrice.Sens.FTC_Ingresso := "A0302_Spintore".IEC.FTC_On;
   "A0302_Manager".CIn.Bordatrice.Sens.FTC_Uscita := "A0302_Bordatrice".IEC_FTC_UscitaBordatrice.FTC_On;

   // TRASFERIMENTO CIn RULLIERA
   "A0302_Manager".CIn.Rulliera.Ax_1 := "A0302_Rulliera".COut.Ax_1;
   "A0302_Manager".CIn.Rulliera.Ax_2 := "A0302_Rulliera".COut.Ax_2;
   "A0302_Manager".CIn.Rulliera.Centraggio := "A0302_Centratori".COut.Centratori;
   "A0302_Manager".CIn.Rulliera.Sollevamento := "A0302_Centratori".COut.Sollevamento;
      // Sensori
   "A0302_Manager".CIn.Rulliera.Coda.Sens.FTC_Rall := "A0302_Rulliera".IEC_FTC_CodaRall.FTC_On;
   "A0302_Manager".CIn.Rulliera.Coda.Sens.FTC_Prox_Ing := "A0302_Rulliera".IEC_FTC_CodaProxIng.FTC_On;
   "A0302_Manager".CIn.Rulliera.Centro.Sens.FTC_Centrale := "A0302_Rulliera".IEC_FTC_Centro.FTC_On;

   // TRASFERIMENTO CIn CARRO PAREGG. CODA
   "A0302_Manager".CIn.CarroPareggCoda.Ax := "A0302_PareggiatoreCoda".COut.Ax;
   "A0302_Manager".CIn.CarroPareggCoda.Ax_InWPos :="A0302_PareggiatoreCoda".COut.Ax_InWPos;
   "A0302_Manager".CIn.CarroPareggCoda.Bloccaggio := "A0302_PareggiatoreCoda".COut.Bloccaggio;
   "A0302_Manager".CIn.CarroPareggCoda.BattutaVerticale := "A0302_PareggiatoreCoda".COut.BattutaVerticale;
   "A0302_Manager".CIn.CarroPareggCoda.PareggiatoreLong := "A0302_PareggiatoreCoda".COut.PareggiatoreLong;
      // Sensori
   "A0302_Manager".CIn.CarroPareggCoda.Sens.FTC_Ingombro_Ing := "A0302_PareggiatoreCoda".IEC_FTC_Input.FTC_On;
   "A0302_Manager".CIn.CarroPareggCoda.Sens.FTC_Ingombro_Out := "A0302_PareggiatoreCoda".IEC_FTC_Output.FTC_On;
   "A0302_Manager".CIn.CarroPareggCoda.Sens.PresenzaMat := "A0302_PareggiatoreCoda".IEC_FTC_PresentMat.FTC_On;
   "A0302_Manager".CIn.CarroPareggCoda.Sens.PosPareggLong.Value := "A0302_PareggiatoreCoda".PosPareggLong.ScaleValue;
   "A0302_Manager".CIn.CarroPareggCoda.Sens.PosPareggLong.Standstill := "A0302_PareggiatoreCoda".PosPareggLong.Standstill;
   "A0302_Manager".CIn.CarroPareggCoda.Sens.PosPareggLong.CheckMeasure := "A0302_PareggiatoreCoda".Ctrl.PareggLong.CheckMesure;

   // TRASFERIMENTO CIn CARRO PAREGG. TESTA
   "A0302_Manager".CIn.CarroPareggTesta.Ax := "A0302_PareggiatoreTesta".COut.Ax;
   "A0302_Manager".CIn.CarroPareggTesta.Ax_InWPos := "A0302_PareggiatoreTesta".COut.Ax_InWPos;
   "A0302_Manager".CIn.CarroPareggTesta.Bloccaggio := "A0302_PareggiatoreTesta".COut.Bloccaggio;
   "A0302_Manager".CIn.CarroPareggTesta.Centraggio := "A0302_PareggiatoreTesta".COut.Centraggio;
   "A0302_Manager".CIn.CarroPareggTesta.Sollevatore := "A0302_PareggiatoreTesta".COut.Sollevatore;
      // Sensori
   "A0302_Manager".CIn.CarroPareggTesta.Sens.FTC_Ingombro_Ing := "A0302_PareggiatoreTesta".IEC_FTC_Rall.FTC_On;
   "A0302_Manager".CIn.CarroPareggTesta.Sens.FTC_Prox_Ls := "A0302_PareggiatoreTesta".IEC_FTC_ProxLs.FTC_On;
   "A0302_Manager".CIn.CarroPareggTesta.Sens.PresenzaMat := "A0302_PareggiatoreTesta".IEC_FTC_PresentMat.FTC_On;

   // TRASFERIMENTO CIn MANIPOLATORI
   // Carro TESTA 
   "A0302_Manager".CIn.Manipolatori.Testa.Ax := "A0302_Manipolatore".COut.Testa.Ax;
   "A0302_Manager".CIn.Manipolatori.Testa.Sollevatore := "A0302_Manipolatore".COut.Testa.Sollevatore;
   "A0302_Manager".CIn.Manipolatori.Testa.Magnete := "A0302_Manipolatore".COut.Testa.Magnete;
   // Carro CODA
   "A0302_Manager".CIn.Manipolatori.Coda.Ax := "A0302_Manipolatore".COut.Coda.Ax;
   "A0302_Manager".CIn.Manipolatori.Coda.Sollevatore := "A0302_Manipolatore".COut.Coda.Sollevatore;
   "A0302_Manager".CIn.Manipolatori.Coda.Magnete := "A0302_Manipolatore".COut.Coda.Magnete;
      // Sensori
   "A0302_Manager".CIn.Manipolatori.InPos_Prelievo := "A0302_Manipolatore".COut.InPos_Prelievo;
   "A0302_Manager".CIn.Manipolatori.InPos_BancoScarto := "A0302_Manipolatore".COut.InPos_BancoScarto;
   "A0302_Manager".CIn.Manipolatori.InPos_BancoA0303 := "A0302_Manipolatore".COut.InPos_BancoA0303;

   // TRASFERIMENTO CIn SPALLE
   "A0302_Manager".CIn.Spalle.Coda.Ax := "Areas_ITF".A04.A0303_SpallaCoda_Cout_Ax;
   "A0302_Manager".CIn.Spalle.Testa.Ax := "Areas_ITF".A04.A0303_SpallaTesta_Cout_Ax;

   // TRASFERIMENTO STATI BANCO A0303
   "A0302_Manager".CIn.Banco_A0303.ReadyToRecive := "Areas_ITF".A04.A0303_Manager_COut_Manipolatore_ReadyToRecive;

   // Production Mng
   "A0302_Manager".CIn.ProdManager := "Areas_ITF".Prod.A03_A04;
END_REGION

REGION Network 3 (SCL): << TRASFERIMENTO stati DataIn del blocco >>
   // MB3 Pulsante semiautomatico 
   "A0302_Manager".DataIn.SemiAut_Pb := "MB3_Pb_Avanti_Stazione_2_Area03";
END_REGION

REGION Network 4 (SCL): << TRASFERIMENTO stati parametri PERS CARRI >>
   // Carro TESTA
   "A0302_PERS".Par.CarroPareggTesta.Preset := "A0302_PareggiatoreTesta_PERS".Par.CarroPareggTesta.Preset;

   // Carro CODA
   "A0302_PERS".Par.CarroPareggCoda.Preset := "A0302_PareggiatoreCoda_PERS".Par.CarroPareggCoda.Preset;

   // Cremaliera
   "A0302_PareggiatoreCoda_PERS".Par.Cremaliera.Modulo := "A0302_PareggiatoreTesta_PERS".Par.Cremaliera.Modulo := "A0302_PERS".Par.Cremaliera.Modulo;
   "A0302_PareggiatoreCoda_PERS".Par.Cremaliera.Passo := "A0302_PareggiatoreTesta_PERS".Par.Cremaliera.Passo := "A0302_PERS".Par.Cremaliera.Passo;
END_REGION

REGION Network 5: << Machine Call >>
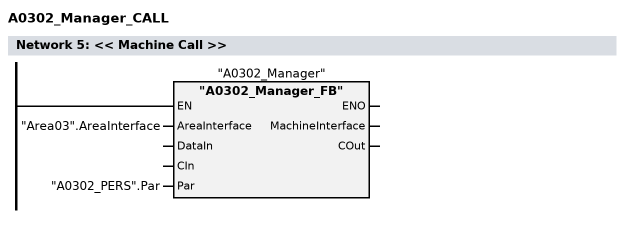
   RUNG wire#powerrail
      "A0302_Manager"(AreaInterface := "Area03".AreaInterface, DataIn :=, CIn :=, Par := "A0302_PERS".Par, MachineInterface =>, COut =>)
   END_RUNG
   // the same network as SCL:
   "A0302_Manager"(AreaInterface := "Area03".AreaInterface, Par := "A0302_PERS".Par);   // "A0302_Manager_FB"
END_REGION
END_FUNCTION

FUNCTION_BLOCK "A0302_Manager_FB"   // FB51, LAD
// stored: MemoryReserve 100, SetENOAutomatically false
   VAR_INPUT
      AreaInterface : "AreaInterface";
      DataIn : Struct
         SemiAut_Pb : Bool;
      END_STRUCT;
      CIn : Struct
         P5 : Struct
            Sollevatori { ExternalAccessible := 'False'; ExternalVisible := 'False'; ExternalWritable := 'False'} : "ValveMachine_COut";
            Spintore_Lat : Struct
               Spin_Lat1 : Struct
                  Standstill : Bool;
                  Rest_CheckNext : Bool;
                  Work_CheckNext : Bool;
                  Rest : Bool;
                  Work : Bool;
               END_STRUCT;
               Spin_Lat2 : Struct
                  Standstill : Bool;
                  Rest_CheckNext : Bool;
                  Work_CheckNext : Bool;
                  Rest : Bool;
                  Work : Bool;
               END_STRUCT;
            END_STRUCT;
            SpintoreLong { ExternalAccessible := 'False'; ExternalVisible := 'False'; ExternalWritable := 'False'} : Struct   // Spintore Longitudinale
               Ax : "Positioning_EPOS_Machine_COut";
               Ax_Sts : Struct
                  PosAttesa_Reached : Bool;
                  PosFineSpinta_Reached : Bool;
               END_STRUCT;
               Spintore : "ValveMachine_COut";
               Vrt : "ValveMachine_COut";
               Orz : "ValveMachine_COut";
               Sens : Struct
                  FTC_FuoriIngombro : Bool;
               END_STRUCT;
            END_STRUCT;
         END_STRUCT;
         Bordatrice : Struct
            Ax : "Positioning_EPOS_Machine_COut";
            Sts : Struct
               PosTargetEnable : Bool;
               PosTarget_Reached : Bool;
               In_W_Pos : Bool;
               AtRest : Bool;
            END_STRUCT;
            Sens : Struct
               FTC_Ingresso : Bool;   // 1833SQ1 - I46.0 (Predisposta - usiamo la 1614BF1)
               FTC_Uscita : Bool;
            END_STRUCT;
         END_STRUCT;
         Rulliera { ExternalAccessible := 'False'; ExternalVisible := 'False'; ExternalWritable := 'False'} : Struct
            Ax_1 : "SpeedMachine_COut";
            Ax_2 : "SpeedMachine_COut";
            Centraggio : "ValveMachine_COut";   // Chiusura Centratori
            Sollevamento : "ValveMachine_COut";   // Solleva centratori
            Coda : Struct
               Sens : Struct
                  FTC_Rall : Bool;   // Sensori presenza materiale banco rallentamento ingresso
                  FTC_Prox_Ing : Bool;   // Sensori presenza materiale banco limite ingresso
               END_STRUCT;
            END_STRUCT;
            Centro : Struct
               Sens : Struct
                  FTC_Centrale : Bool;
               END_STRUCT;
            END_STRUCT;
         END_STRUCT;
         CarroPareggCoda { ExternalAccessible := 'False'; ExternalVisible := 'False'; ExternalWritable := 'False'} : Struct
            Ax_InWPos : Bool;
            Ax : "Positioning_DOL_Machine_COut";
            Bloccaggio : "ValveMachine_COut";
            BattutaVerticale : "ValveMachine_COut";
            PareggiatoreLong : "ValveMachine_COut";
            Sens : Struct
               FTC_Ingombro_Ing : Bool;   // FTC fuori ingombro lato ingresso al carro pareggiatore di coda
               FTC_Ingombro_Out : Bool;   // FTC fuori ingombro lato uscita al carro pareggiatore di coda
               PresenzaMat : Bool;   // FC presenza materiale agganciato
               PosPareggLong : Struct
                  Value : LReal;
                  CheckMeasure : Bool;
                  Standstill : Bool;
               END_STRUCT;
            END_STRUCT;
         END_STRUCT;
         CarroPareggTesta { ExternalAccessible := 'False'; ExternalVisible := 'False'; ExternalWritable := 'False'} : Struct
            Ax_InWPos : Bool;
            Ax : "Positioning_DOL_Machine_COut";
            Bloccaggio : "ValveMachine_COut";
            Centraggio : "ValveMachine_COut";
            Sollevatore : "ValveMachine_COut";
            Sens : Struct
               FTC_Ingombro_Ing : Bool;   // FTC fuori ingombro lato ingresso al carro pareggiatore di testa - Rallentamento rulliera
               FTC_Prox_Ls : Bool;   // FTC sensore presenza materiale banco limite ingresso
               PresenzaMat : Bool;   // FC presenza materiale agganciato
            END_STRUCT;
         END_STRUCT;
         Manipolatori : Struct
            Testa : Struct
               Ax : "Positioning_EPOS_Machine_COut";
               Sollevatore : "ValveMachine_COut";
               Magnete : "ValveMachine_COut";
            END_STRUCT;
            Coda : Struct
               Ax : "Positioning_EPOS_Machine_COut";
               Sollevatore : "ValveMachine_COut";
               Magnete : "ValveMachine_COut";
            END_STRUCT;
            InPos_Prelievo : Bool;
            InPos_BancoScarto : Bool;
            InPos_BancoA0303 : Bool;
         END_STRUCT;
         Spalle : Struct
            Coda : Struct
               Ax : "Positioning_DOL_Machine_COut";
            END_STRUCT;
            Testa : Struct
               Ax : "Positioning_DOL_Machine_COut";
            END_STRUCT;
         END_STRUCT;
         Banco_A0303 : Struct
            ReadyToRecive : Bool;   // Consenso da Stazione A0303 a ricevere il pezzo buono misurato
         END_STRUCT;
         ProdManager : "Prod_Beam_Ctrl";
      END_STRUCT;
   END_VAR
   VAR_OUTPUT
      MachineInterface : "MachineInterface";
      COut : Struct
         HU : Struct
            EnableStopDoorOpeningReq : Bool;
            EnableStopInPhase : Bool;
            EnableStopProgrammed : Bool;
            Control_ON : Bool;
            Rest : Bool;
            Work : Bool;
         END_STRUCT;
         SpintoreLong : Struct
            EnableStopDoorOpeningReq : Bool;
            EnableStopInPhase : Bool;
            EnableStopProgrammed : Bool;
            Control_ON : Bool;
            REST_Req : Bool;
            WORK_Req : Bool;
            Rest : Bool;
            Work : Bool;
         END_STRUCT;
         Bordatrice : Struct
            Ax : "Positioning_EPOS_Machine_Manager";
            Sts : Struct
               PosTarget_Reached : Bool;
               AtRest : Bool;
            END_STRUCT;
            DataOut : "Positioning_EPOS_Machine_DataOut";
            Rest_Req : Bool;
            Work_Req : Bool;
         END_STRUCT;
         Rulliera : Struct
            Ax_1 : "SpeedMachine_CIn_Manager";
            Ax_2 : "SpeedMachine_CIn_Manager";
            Centratori : Struct   // Chiusura Centratori
               Sollevamento : "ValveMachine_Manager";
               Centraggio : "ValveMachine_Manager";
            END_STRUCT;
            Ax_1_Frw_Req : Bool;
            Ax_1_Brw_Req : Bool;
            Ax_2_Frw_Req : Bool;
            Ax_2_Brw_Req : Bool;
         END_STRUCT;
         CarroPareggCoda : Struct
            EnableStopDoorOpeningReq : Bool;
            EnableStopInPhase : Bool;
            EnableStopProgrammed : Bool;
            Control_ON : Bool;
            MoveToPos : Bool;
            Pos : LReal;
            Speed : LReal;
            Bloccaggio : Struct
               Rest : Bool;
               Work : Bool;
            END_STRUCT;
            BattutaVrt : Struct
               Rest : Bool;
               Work : Bool;
            END_STRUCT;
            PareggLong : Struct
               Rest : Bool;
               Work : Bool;
            END_STRUCT;
         END_STRUCT;
         CarroPareggTesta : Struct
            EnableStopDoorOpeningReq : Bool;
            EnableStopInPhase : Bool;
            EnableStopProgrammed : Bool;
            Control_ON : Bool;
            MoveToPos : Bool;
            Pos : LReal;
            Speed : LReal;
            Bloccaggio : "OP_PB";
            Sollevamento : "OP_PB";
            Centraggio : "OP_PB";
         END_STRUCT;
         Manipolatori : Struct
            Ax : Struct
               EnableStopDoorOpeningReq : Bool;
               EnableStopInPhase : Bool;
               EnableStopProgrammed : Bool;
               Control_ON : Bool;
               MoveToPos : Bool;
               Pos : LReal;
               Vel : LReal;
               Acc : LReal;
               Dec : LReal;
            END_STRUCT;
            Sollevatori : "OP_PB";
            Magneti : "OP_PB";
         END_STRUCT;
      END_STRUCT;
   END_VAR
   VAR_IN_OUT
      Par : Struct
         CarroPareggCoda : Struct
            Delay_StartMove : Time;
            Preset : LReal;
         END_STRUCT;
         CarroPareggTesta : Struct
            Delay_StartMove : Time;
            Preset : LReal;
         END_STRUCT;
         Cremaliera : Struct
            Modulo : LReal;
            Passo : LReal;
         END_STRUCT;
      END_STRUCT;
   END_VAR
   VAR
      Alarm : Struct
         Qlty_Unknow : Bool;   // Allarme pezzo sconosciuto
         ToCheckList_Full : Bool;
         WrongReadPz_ManipBasso : Bool;
         Pz_NonPareggiabile : Bool;
         STOP_FineTurno : Bool;
         STOP_End_Of_Proroduction : Bool;
         STOP_ControlloQualita : Bool;
      END_STRUCT;
      Warning : Struct
         CheckBancoAccumulo : Bool;
      END_STRUCT;
      Sts : Struct
         SemiAut : Struct
            ON : Bool;
            Request : Bool;
            MaterialFrw : Bool;
         END_STRUCT;
         CarroPareggTesta : Struct
            InCyclePos : Bool;
         END_STRUCT;
         CarroPareggCoda : Struct
            InCyclePos : Bool;
         END_STRUCT;
         Attrezzamento : Struct
            Ready : Bool;
            FindNewID : Bool;
            RequestNewPosition : Bool;
            OLD_OID : DInt;
         END_STRUCT;
         BTrk : Struct
            A0302Exit_Actual_O_ID : DInt;
            BLen_Paregg : Real;
            Last_Misure1Paregg : Real;
            Last_Misure2Paregg : Real;
            A0302Entry_Absence : Bool;
            A0302Exit_Absence : Bool;
            ZoneA0302Entry_Empty : Bool;
            ZoneA0302Exit_Empty : Bool;
            A0302_CheckBancoAccumulo : Bool;
            Waiting_A0302_Recive : Bool;
         END_STRUCT;
         AlarmsPresence : Bool;
         WarningsPresence : Bool;
         IsStandstill : Bool;
      END_STRUCT;
      Ctrl : Struct
         Stop : Bool;
         TRK : Struct
            BTrk : Struct
               "P5.1_To_LongPosAttesa" : Bool;
               "P5.2_LongPosAttesa_TO_Spintore" : Bool;
               "P5.2_Spintore_TO_ExitA031" : Bool;
               "P5.2_ExitA031_To_IngBord" : Bool;
               "P5.2_Ax_MoveToPosAttesa" : Bool;
               "P5.2_Ax_PreparingPosAttesa" : Bool;
               "P5.2_Ax_MoveToPosSpinta" : Bool;
               SpinBord_In_To_Bord_In : Bool;
               Bordatrice_In_To_Out : Bool;   // il pezzo ha raggiunto il sensore di uscita della bordatrice (xxxSQx) (salvataggio posizione asse bordatrice)
               Bordatrice_Out_To_PareggCodaUp : Bool;   // Il pezzo è in uscita della bordatrice e la posizione target non è limitata perchè il pareggiamento di coda è alto
               Bordatrice_Out_To_PareggCodaDown : Bool;   // Il pezzo è in uscita della bordatrice ma la posizione target è limitata per non collidere con il pareggiamento di coda basso
               Rulliera_Start_Brw : Bool;
               Rulliera_Ax_1_Start_Frw : Bool;
               Rulliera_Ax_2_Start_Frw : Bool;
               RulliereVode : Bool;
               PCodaDown_TO_Rulli_PCodaDown : Bool;   // Pezzo su rulliera (1) + pareggiatore coda basso quindi quando incontra sensore (1,2) deve rallentare
               PCodaDown_TO_RALL_Rulli_PCodaDown : Bool;   // Pezzo su rulliera (1) + pareggiatore coda basso e ha incontrato sensore (1,2) di rallentamento
               PCodaDown_TO_STOP_PCodaDown : Bool;   // Pezzo su rulliera (1) + pareggiatore coda basso e ha incontrato sensore (3) di stop
               STOP_PCodaDown_TO_PCoda_Up : Bool;   // Pezzo su rulliera (1) + pareggiatore coda alto quindi può muoversi liberamente
               "PareggCodaUp_To_Rull-PrimaPareggCodaAltro" : Bool;
               PCoda_Up_TO_PCoda_UP_S3 : Bool;   // Pezzo su rulliera (1) + pareggiatore coda alto ed ha incontrato il sensore 3 (in ingresso al pareg.)
               PCoda_UP_S3_TO_PCoda_UP_S4 : Bool;   // Pezzo su rulliera (1) + pareggiatore coda alto ed ha incontrato il sensore 4 (in uscita al pareg.)
               PCoda_UP_S4_TO_PCoda_DownCnd : Bool;   // Pezzo su rulliera (1/2) + pareggiatore coda che è alto ed ha liberato il sensore 4-> Pareg. può andare basso (posizione di lavoro)
               PCoda_Beam_TO_PTesta : Bool;   // Pezzo su rulliera (1/2) tra il pareggiatore di testa e quello di coda
               Beam_TO_Stop_PTesta : Bool;   // Pezzo su rulliera (1/2) + ha incontrato il sensore 5 su pareggiatore di testa
               "Stop_PTesta_TO_Rull-Centratori" : Bool;   // Pezzo su rulliera (1/2) tra i pareggiatori + centratori a lavoro
               "Rull-Centratori_TO_Cnd_PareggCoda" : Bool;   // Pezzo su rulliera (1/2) tra i pareggiatori (quello di coda è basso) + centratori a lavoro
               Cnd_PareggCoda_TO_Pareggiato : Bool;   // Pezzo su rulliera (1/2) tra i pareggiatori e paregiatura di coda eseguito lavoro cilindro idraulico (ora si sa la misura del pezzo, si può mettere utenze in attesa del prossimo pezzo)
               Check_Tolleranza_BLen_Qlty : Bool;
               Pareggiato_TO_PresaBasso : Bool;   // Pezzo su magneti del manipolatore basso in posizione di presa.
               PresaBasso_TO_PresaAlto : Bool;   // Pezzo su magneti del manipolatore alto in posizione di presa.
               PresaAlto_To_CheckOut_BadQlty : Bool;   // Pezzo su magneti del manipolatore alto in posizione di uscita perchè non conforme
               CheckOut_BadQlty_UP_MoveToPos : Bool;   // Ho il pezzo in presa alta > vado in posizione uscita banco scarto
               PresaAlto_To_CheckOut_GoodQlty : Bool;   // Pezzo su magneti del manipolatore alto in posizione per deposito su A0303
               CheckOut_GoodQlty_UP_MoveToPos : Bool;   // Ho il pezzo in presa alta > vado in posizione uscita banco A0303
               CheckOut_BadQlty_UP_To_DOWN : Bool;   // Pezzo su magneti del manipolatore basso in posizione di uscita perchè non conforme
               CheckOut_BadQlty_DOWN_To_Sgancia : Bool;
               CheckOut_GoodQlty_UP_To_DOWN : Bool;   // Pezzo su magneti del manipolatore basso in posizione per deposito su A0303
               CheckOut_GoodQlty_DOWN_To_Sgancia : Bool;
               Manipolatori_Return_ToPrelievo : Bool;   // Ritorno degli assi manipolatore a zero e / o a prelievo
            END_STRUCT;
            BTrk_ToCheck : Struct
               ClearList : Bool;
               QtyClear_RetVal : Bool;
               Prelievo_RecondGood : Bool;   // Attivo durante la fase di posizionamento manuale del Beam fino a quando il manipolatore lo prende
               RecG_InPos_Centraggio : Bool;   // Beam ricondizionato posizionato su rulliera da centrare
               RegG_InPos_ReadyPickUp : Bool;
            END_STRUCT;
         END_STRUCT;
         SpintoreLong : Struct
            Rest : Bool;
            Work : Bool;
            MoveAttesaDisable : Bool;
         END_STRUCT;
         Bordatrice : Struct
            Run : Bool;
         END_STRUCT;
         Rulliera : Struct
            Ax_1_Vel_Bord : Bool;
            Ax_2_Vel_Bord : Bool;
            Ax_1_Lenta_CarroCoda : Bool;
            Ax_1_2_Vel_CarroTesta : Bool;
            Ax_1_2_Vel_ZeroTesta : Bool;
            Ax_1_2_Vel_Appoggio : Bool;
            Ax_1_2_End_VelZero : Bool;
            Ax_2_MemoRall : Bool;
            SP_TimeMemoRall : Time;
            TON_RitardoRallenta : IEC_TIMER;
            Centraggio : Struct
               Rest : Bool;
               Work : Bool;
            END_STRUCT;
            Sollevamento : Struct
               Rest : Bool;
               Work : Bool;
            END_STRUCT;
         END_STRUCT;
         CarroPareggCoda : Struct
            Ax : Struct
               MoveToPos : Bool;
               Pos : LReal;
            END_STRUCT;
            Bloccaggio : Struct
               Rest : Bool;
               Work : Bool;
            END_STRUCT;
            BattutaVerticale : Struct
               Rest : Bool;
               Work : Bool;
            END_STRUCT;
            PareggiatoreLong : Struct
               Rest : Bool;
               Work : Bool;
            END_STRUCT;
            MisuraPzPareggiato : Bool;
         END_STRUCT;
         CarroPareggTesta : Struct
            Ax : Struct
               MoveToPos : Bool;
               Pos : LReal;
            END_STRUCT;
            Bloccaggio : Struct
               Rest : Bool;
               Work : Bool;
            END_STRUCT;
            Sollevatore : Struct
               Rest : Bool;
               Work : Bool;
            END_STRUCT;
            Centraggio : Struct
               Rest : Bool;
               Work : Bool;
            END_STRUCT;
         END_STRUCT;
         Manipolatori : Struct
            Ax : Struct
               MoveToPos : Bool;
               Pos : LReal;
            END_STRUCT;
            Sollevatori : Struct
               Rest : Bool;
               Work : Bool;
            END_STRUCT;
            Magneti : Struct
               Rest : Bool;
               Work : Bool;
            END_STRUCT;
         END_STRUCT;
      END_STRUCT;
      HMI : Struct
         PlsClear_ListToCheck : Bool;
      END_STRUCT;
      BTrk_A0302_Exit_Item : Struct
         BLean : Real;
         W_A : Real;
         Tol_Max : Real;
         Tol_Min : Real;
         Good { ExternalAccessible := 'False'; ExternalVisible := 'False'; ExternalWritable := 'False'} : Bool;
         ToCheckLen { ExternalAccessible := 'False'; ExternalVisible := 'False'; ExternalWritable := 'False'} : Bool;
      END_STRUCT;
      BTrk_ListToCheck : Struct
         Recond : Struct
            Found : Bool;
            Nr_B : Int;
         END_STRUCT;
      END_STRUCT;
      OffsetCarri : Struct
         DaSpallaTesta : LReal;
         DaSpallaCoda : LReal;
      END_STRUCT;
      CarroTesta : Struct
         RimanenzaPos : LReal;
         PassoReq : LReal;
         PosBattutePz : LReal;
         SemiBeamLen : LReal;
         NrPassiReq : LReal;
      END_STRUCT;
      CarroCoda : Struct
         RimanenzaPos : LReal;
         PassoReq : LReal;
         PosBattutePz : LReal;
         SemiBeamLen : LReal;
         NrPassiReq : LReal;
      END_STRUCT;
      TON_AlarmWrongReadPz_Manip : IEC_TIMER;
      TON_Alarm_FTC_CarroCodaOut { S7_SetPoint := 'True'} : IEC_TIMER;
      TON_Stop { S7_SetPoint := 'True'} : IEC_TIMER;
   END_VAR
   VAR_TEMP
      AUX : Struct
         SemiAut_Pb : Bool;
      END_STRUCT;
      i : Int;
      BTrk_A0302_EXIT_GetData : Struct   // Appoggio struttura per lettura dati dal Mes
         indx : Int;   // Se trovato tra i TODO / ENDING / OUT questo è l'indice dove sono stati prelevati i dati
         Sts : Int;   // 0 = Non Trovato; 0 = ACT; 1 = TODO; 2=ENDING; 3 = OUT
         Item : "Prod_Item_small";
      END_STRUCT;
      DisableA0302 : Bool;
      PieceToCheck_Presence : Bool;
      CarroTestaCentraggio_Disable : Bool;
   END_VAR
   VAR CONSTANT
      OffsetGioco : Real := 2.0;   // Offset gioco carri durante lettura Pareggiamento pezzo
   END_VAR
   VAR_TEMP   // added for the SCL form of the ladder/FBD networks
      _w1 : Bool;
      _w2 : Bool;
      _w3 : Bool;
      _w4 : Bool;
      _w5 : Bool;
      _w6 : Bool;
      _w7 : Bool;
      _w8 : Bool;
      _w9 : Bool;
      _w10 : Bool;
      _w11 : Bool;
      _w12 : Bool;
      _w13 : Bool;
      _w14 : Bool;
      _w15 : Bool;
      _w16 : Bool;
      _w17 : Bool;
      _w18 : Bool;
      _w19 : Bool;
      _w20 : Bool;
   END_VAR
BEGIN

REGION Network 1 (SCL): = Area - Rst =
   IF #AreaInterface.RstAlarms THEN
       #Alarm.Qlty_Unknow := FALSE;
       #Alarm.ToCheckList_Full := FALSE;
       #Alarm.STOP_ControlloQualita := FALSE;
       #Alarm.STOP_FineTurno := FALSE;
       #Alarm.STOP_End_Of_Proroduction := FALSE;
   END_IF;

   IF #AreaInterface.RstAlarms AND #CIn.CarroPareggCoda.Sens.PresenzaMat AND #CIn.CarroPareggTesta.Sens.PresenzaMat
       AND #CIn.Manipolatori.Testa.Magnete.Work AND #CIn.Manipolatori.Coda.Magnete.Work THEN
       #Alarm.WrongReadPz_ManipBasso := FALSE;
   END_IF;

   IF #AreaInterface.RstAlarms AND NOT #CIn.CarroPareggCoda.Sens.FTC_Ingombro_Out THEN
       #Alarm.Pz_NonPareggiabile := FALSE;
   END_IF;
END_REGION

REGION Network 2: ******** CLEAR TRACKING ARRIVATO ********
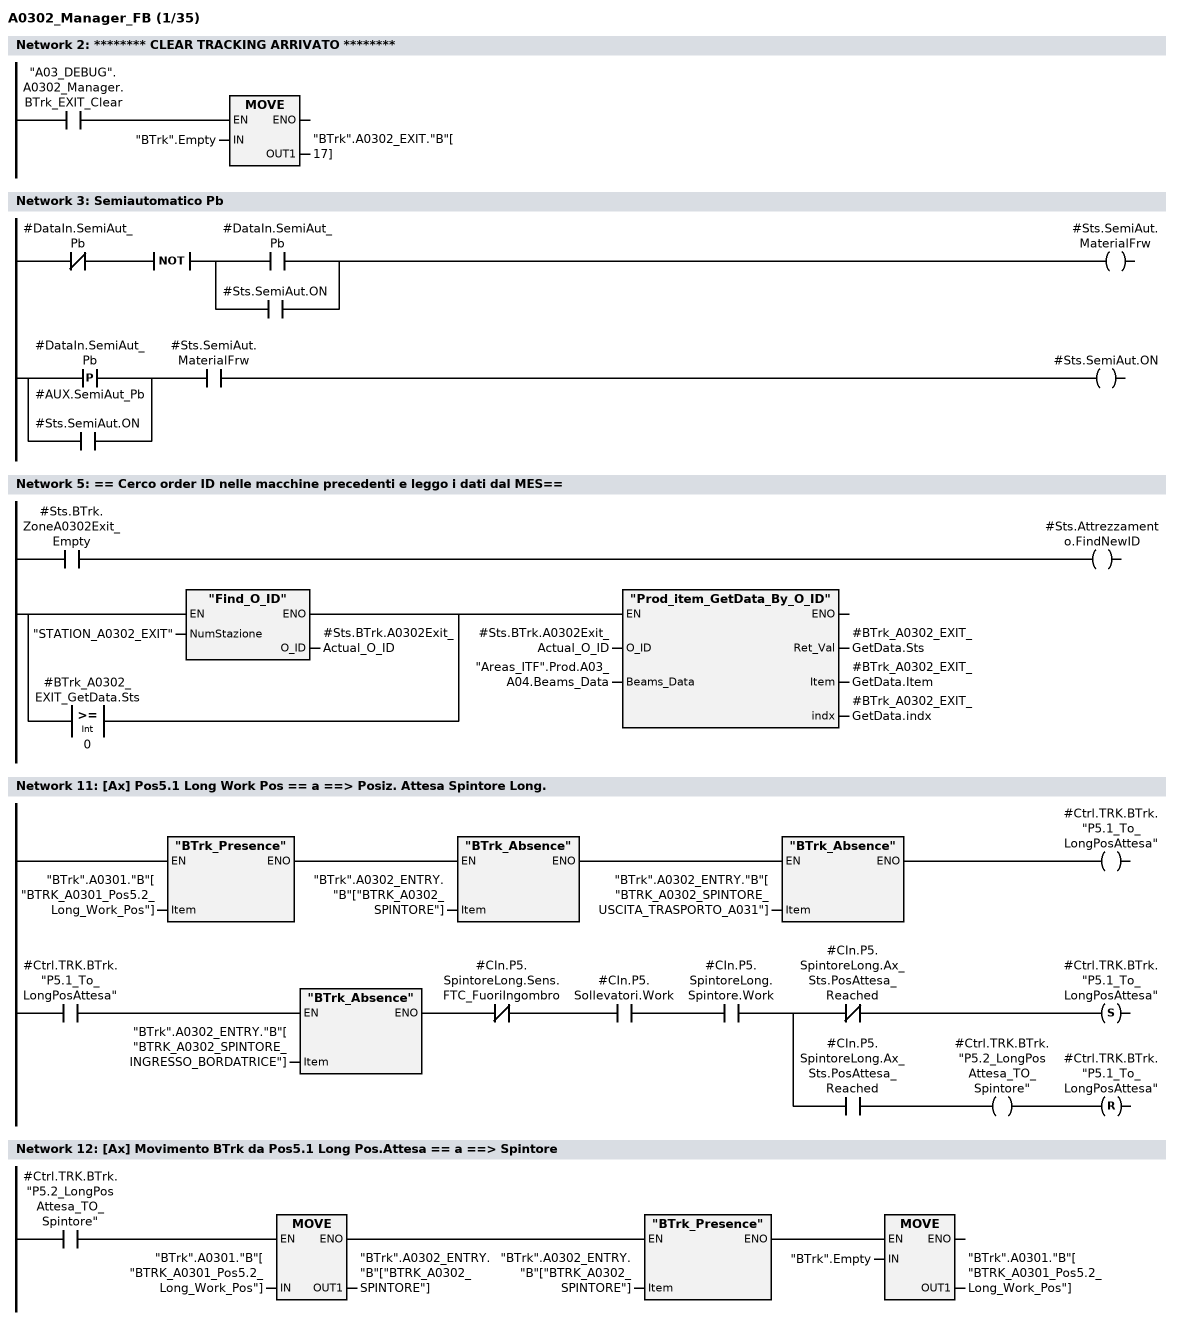
   RUNG wire#powerrail
      Contact( "A03_DEBUG".A0302_Manager.BTrk_EXIT_Clear )
      Move(in := "BTrk".Empty, out1 => "BTrk".A0302_EXIT."B"[17])
   END_RUNG
   // the same network as SCL:
   IF "A03_DEBUG".A0302_Manager.BTrk_EXIT_Clear THEN "BTrk".A0302_EXIT."B"[17] := "BTrk".Empty; END_IF;
END_REGION

REGION Network 3: Semiautomatico Pb
   RUNG wire#powerrail
      I_Contact( #DataIn.SemiAut_Pb )
      Not()
      wire#w1
      Contact( #DataIn.SemiAut_Pb )
      wire#w2
      Coil( #Sts.SemiAut.MaterialFrw )
   END_RUNG
   RUNG wire#w1
      Contact( #Sts.SemiAut.ON )
   END_RUNG wire#w2
   RUNG wire#powerrail
      P_Contact(operand := #DataIn.SemiAut_Pb, bit := #AUX.SemiAut_Pb)
      wire#w3
      Contact( #Sts.SemiAut.MaterialFrw )
      Coil( #Sts.SemiAut.ON )
   END_RUNG
   RUNG wire#powerrail
      Contact( #Sts.SemiAut.ON )
   END_RUNG wire#w3
   // the same network as SCL:
   #Sts.SemiAut.MaterialFrw := NOT (NOT #DataIn.SemiAut_Pb) AND (#DataIn.SemiAut_Pb OR #Sts.SemiAut.ON);
   #_w1 := #DataIn.SemiAut_Pb AND NOT #AUX.SemiAut_Pb;   // rising edge of #DataIn.SemiAut_Pb
   #AUX.SemiAut_Pb := #DataIn.SemiAut_Pb;
   #Sts.SemiAut.ON := (#_w1 OR #Sts.SemiAut.ON) AND #Sts.SemiAut.MaterialFrw;
END_REGION

REGION Network 5: == Cerco order ID nelle macchine precedenti e leggo i dati dal MES==
   RUNG wire#powerrail
      Contact( #Sts.BTrk.ZoneA0302Exit_Empty )
      Coil( #Sts.Attrezzamento.FindNewID )
   END_RUNG
   RUNG wire#powerrail
      "Find_O_ID"(NumStazione := "STATION_A0302_EXIT", O_ID => #Sts.BTrk.A0302Exit_Actual_O_ID)
      wire#w1
      "Prod_item_GetData_By_O_ID"(O_ID := #Sts.BTrk.A0302Exit_Actual_O_ID, Beams_Data := "Areas_ITF".Prod.A03_A04.Beams_Data, Ret_Val => #BTrk_A0302_EXIT_GetData.Sts, Item => #BTrk_A0302_EXIT_GetData.Item, indx => #BTrk_A0302_EXIT_GetData.indx)
   END_RUNG
   RUNG wire#powerrail
      { S7_Templates := "SrcType := Int" } GE_Contact(in1 := #BTrk_A0302_EXIT_GetData.Sts, in2 := 0)
   END_RUNG wire#w1
   // the same network as SCL:
   #Sts.Attrezzamento.FindNewID := #Sts.BTrk.ZoneA0302Exit_Empty;
   "Find_O_ID"(NumStazione := "STATION_A0302_EXIT", O_ID => #Sts.BTrk.A0302Exit_Actual_O_ID, ENO => #_w1);
   IF #_w1 OR (#BTrk_A0302_EXIT_GetData.Sts >= 0) THEN
       #BTrk_A0302_EXIT_GetData.Sts := "Prod_item_GetData_By_O_ID"(O_ID := #Sts.BTrk.A0302Exit_Actual_O_ID,
                               Beams_Data := "Areas_ITF".Prod.A03_A04.Beams_Data,
                               Item => #BTrk_A0302_EXIT_GetData.Item,
                               indx => #BTrk_A0302_EXIT_GetData.indx);
   END_IF;
END_REGION

REGION Network 6 (SCL): == Richiesta nuovo posizionamento carri Testa/Coda per cambio Traking ==

   //Se ho O_ID <> e non sono vuoto attivo avviso di attesa zona A0302 vuota
   IF (#Sts.BTrk.A0302Exit_Actual_O_ID <> #Sts.Attrezzamento.OLD_OID) OR (NOT #Sts.BTrk.ZoneA0302Exit_Empty OR NOT #Sts.BTrk.ZoneA0302Entry_Empty)THEN
       #Sts.BTrk.Waiting_A0302_Recive := TRUE;

   ELSIF (#Sts.BTrk.A0302Exit_Actual_O_ID = #Sts.Attrezzamento.OLD_OID) OR ( #Sts.BTrk.ZoneA0302Exit_Empty AND #Sts.BTrk.ZoneA0302Entry_Empty) THEN
       #Sts.BTrk.Waiting_A0302_Recive := FALSE;

   END_IF;

   //Se ho O_ID <> e sono vuoto aggiorno vecchio O_ID 
   IF (#Sts.BTrk.A0302Exit_Actual_O_ID <> #Sts.Attrezzamento.OLD_OID) AND #Sts.BTrk.ZoneA0302Exit_Empty AND #Sts.BTrk.ZoneA0302Entry_Empty THEN
       #Sts.Attrezzamento.OLD_OID := #Sts.BTrk.A0302Exit_Actual_O_ID;
   END_IF;
END_REGION

REGION Network 7 (SCL): == Compilo i dati del btrk in base all'order ID in arrivo ==

   IF #BTrk_A0302_EXIT_GetData.Sts >= 0 THEN

       "BTrk".A0302_EXIT.O_ID:="BTrk".A0302_ENTRY.O_ID := #Sts.Attrezzamento.OLD_OID;
       "BTrk".A0302_EXIT.Beam_Len := "BTrk".A0302_ENTRY.Beam_Len := #BTrk_A0302_EXIT_GetData.Item.Beams_Len;
       "BTrk".A0302_EXIT.Beam_W_A := "BTrk".A0302_ENTRY.Beam_W_A := #BTrk_A0302_EXIT_GetData.Item.Beams_W_A;
       "BTrk".A0302_EXIT.Beam_H_B := "BTrk".A0302_ENTRY.Beam_H_B := #BTrk_A0302_EXIT_GetData.Item.Beams_H_B;

   ELSE
           "BTrk".A0302_EXIT.O_ID := "BTrk".A0302_ENTRY.O_ID := "BTrk".A0301.O_ID := -1;
           "BTrk".A0302_EXIT.Beam_Len := "BTrk".A0302_ENTRY.Beam_Len := -1.0;
           "BTrk".A0302_EXIT.Beam_W_A := "BTrk".A0302_ENTRY.Beam_W_A := -1.0;
           "BTrk".A0302_EXIT.Beam_H_B := "BTrk".A0302_ENTRY.Beam_H_B := -1.0;
   END_IF;
END_REGION

REGION Network 8 (SCL): == Richiesta nuovo posizionamento x cambio Order ID ==

   #Sts.Attrezzamento.RequestNewPosition := ("BTrk".A0302_EXIT.O_ID <> -1)
   AND (#BTrk_A0302_EXIT_GetData.Sts >= 0)
   AND (#BTrk_A0302_EXIT_GetData.Item.Beam_Code = 1)
   AND #Sts.Attrezzamento.FindNewID
   AND NOT #Sts.Attrezzamento.Ready
   AND NOT #BTrk_ListToCheck.Recond.Found
   AND (NOT #CIn.CarroPareggCoda.Ax_InWPos OR NOT #CIn.CarroPareggTesta.Ax_InWPos);
END_REGION

REGION Network 10: <<<< SPINTORE LONGITUDINALE >>>>
END_REGION

REGION Network 11: [Ax] Pos5.1 Long Work Pos == a ==> Posiz. Attesa Spintore Long.
   RUNG wire#powerrail
      "BTrk_Presence"(Item := "BTrk".A0301."B"["BTRK_A0301_Pos5.2_Long_Work_Pos"])
      "BTrk_Absence"(Item := "BTrk".A0302_ENTRY."B"["BTRK_A0302_SPINTORE"])
      "BTrk_Absence"(Item := "BTrk".A0302_ENTRY."B"["BTRK_A0302_SPINTORE_USCITA_TRASPORTO_A031"])
      Coil( #Ctrl.TRK.BTrk."P5.1_To_LongPosAttesa" )
   END_RUNG
   RUNG wire#powerrail
      Contact( #Ctrl.TRK.BTrk."P5.1_To_LongPosAttesa" )
      "BTrk_Absence"(Item := "BTrk".A0302_ENTRY."B"["BTRK_A0302_SPINTORE_INGRESSO_BORDATRICE"])
      I_Contact( #CIn.P5.SpintoreLong.Sens.FTC_FuoriIngombro )
      Contact( #CIn.P5.Sollevatori.Work )
      Contact( #CIn.P5.SpintoreLong.Spintore.Work )
      wire#w1
      I_Contact( #CIn.P5.SpintoreLong.Ax_Sts.PosAttesa_Reached )
      S_Coil( #Ctrl.TRK.BTrk."P5.1_To_LongPosAttesa" )
   END_RUNG
   RUNG wire#w1
      Contact( #CIn.P5.SpintoreLong.Ax_Sts.PosAttesa_Reached )
      Coil( #Ctrl.TRK.BTrk."P5.2_LongPosAttesa_TO_Spintore" )
      R_Coil( #Ctrl.TRK.BTrk."P5.1_To_LongPosAttesa" )
   END_RUNG
   // the same network as SCL:
   "BTrk_Presence"(Item := "BTrk".A0301."B"["BTRK_A0301_Pos5.2_Long_Work_Pos"], ENO => #_w1);
   "BTrk_Absence"(EN := #_w1, Item := "BTrk".A0302_ENTRY."B"["BTRK_A0302_SPINTORE"], ENO => #_w2);
   "BTrk_Absence"(EN := #_w2,
                  Item := "BTrk".A0302_ENTRY."B"["BTRK_A0302_SPINTORE_USCITA_TRASPORTO_A031"],
                  ENO => #_w3);
   #Ctrl.TRK.BTrk."P5.1_To_LongPosAttesa" := #_w3;
   "BTrk_Absence"(EN := #Ctrl.TRK.BTrk."P5.1_To_LongPosAttesa",
                  Item := "BTrk".A0302_ENTRY."B"["BTRK_A0302_SPINTORE_INGRESSO_BORDATRICE"],
                  ENO => #_w4);
   #_w5 := #_w4 AND NOT #CIn.P5.SpintoreLong.Sens.FTC_FuoriIngombro AND #CIn.P5.Sollevatori.Work AND #CIn.P5.SpintoreLong.Spintore.Work;
   IF #_w5 AND NOT #CIn.P5.SpintoreLong.Ax_Sts.PosAttesa_Reached THEN
       #Ctrl.TRK.BTrk."P5.1_To_LongPosAttesa" := TRUE;
   END_IF;
   #Ctrl.TRK.BTrk."P5.2_LongPosAttesa_TO_Spintore" := #_w5 AND #CIn.P5.SpintoreLong.Ax_Sts.PosAttesa_Reached;
   IF #Ctrl.TRK.BTrk."P5.2_LongPosAttesa_TO_Spintore" THEN
       #Ctrl.TRK.BTrk."P5.1_To_LongPosAttesa" := FALSE;
   END_IF;
END_REGION

REGION Network 12: [Ax] Movimento BTrk da Pos5.1 Long Pos.Attesa == a ==> Spintore
   RUNG wire#powerrail
      Contact( #Ctrl.TRK.BTrk."P5.2_LongPosAttesa_TO_Spintore" )
      Move(in := "BTrk".A0301."B"["BTRK_A0301_Pos5.2_Long_Work_Pos"], out1 => "BTrk".A0302_ENTRY."B"["BTRK_A0302_SPINTORE"])
      "BTrk_Presence"(Item := "BTrk".A0302_ENTRY."B"["BTRK_A0302_SPINTORE"])
      Move(in := "BTrk".Empty, out1 => "BTrk".A0301."B"["BTRK_A0301_Pos5.2_Long_Work_Pos"])
   END_RUNG
   // the same network as SCL:
   IF #Ctrl.TRK.BTrk."P5.2_LongPosAttesa_TO_Spintore" THEN
       "BTrk".A0302_ENTRY."B"["BTRK_A0302_SPINTORE"] := "BTrk".A0301."B"["BTRK_A0301_Pos5.2_Long_Work_Pos"];
   END_IF;
   "BTrk_Presence"(EN := #Ctrl.TRK.BTrk."P5.2_LongPosAttesa_TO_Spintore",
                   Item := "BTrk".A0302_ENTRY."B"["BTRK_A0302_SPINTORE"],
                   ENO => #_w1);
   IF #_w1 THEN "BTrk".A0301."B"["BTRK_A0301_Pos5.2_Long_Work_Pos"] := "BTrk".Empty; END_IF;
END_REGION

